# B&R Automation Studio project 305841_E00002_AM_0 (part 8)

#### ActionMotionFbs.st
```iecst
(********************************************************************
 * COPYRIGHT -- General Atomics
 ********************************************************************
 * Program: AxisStateMachine
 * File: ActionMoveVel.st
 * Author: Administrator
 * Created: January 22, 2014
 ********************************************************************
 * Implementation of program AxisStateMachine
 ********************************************************************)

ACTION ActionCallMotionFunctions:
  ActionMpAxisBasic;
  ActionCamInOut;
  ActionGearInOut;
  ActionOffsetShift;
  ActionPhaseShift;
END_ACTION

ACTION ActionMpAxisBasic:
  // 1) Range checks position, velocity, accel & Decel
  // 2) Packs the sMot_MoveParameters into a local axisBasicParamsStructure
  // 3) Detects parameter changes and manages the Update and UpdateDone bits
  // 4) Sets the fb command bits based on the axis sMot_AxisCommands structure
  // 5) Runs the fbMpAxisBasic funciton block
  // 6) Updates the axis structure with the status and axis info coming back from the fb

  // Make sure min/max values are not exceeded for position, velocity, accel, and decel.
  // Clamp if necessary

  // Position
  IF ax.MoveParameters.Position >  axPositionLimits.PositionLimitPos THEN
    ax.MoveParameters.Position :=  axPositionLimits.PositionLimitPos;
  END_IF;
  IF ax.MoveParameters.Position <  axPositionLimits.PositionLimitNeg THEN
    ax.MoveParameters.Position :=  axPositionLimits.PositionLimitNeg;
  END_IF;

  // Velocity
  IF ax.MoveParameters.Velocity > ax.MoveParameters.VelocityMax THEN
    ax.MoveParameters.Velocity := ax.MoveParameters.VelocityMax;
  END_IF;
  IF ax.MoveParameters.Velocity < ax.MoveParameters.VelocityMin THEN
    ax.MoveParameters.Velocity := ax.MoveParameters.VelocityMin;
  END_IF;

  // Accel and decel
  IF ax.MoveParameters.Acceleration > ax.MoveParameters.AccelMax THEN
    ax.MoveParameters.Acceleration := ax.MoveParameters.AccelMax;
  END_IF;
  IF ax.MoveParameters.Acceleration < ax.MoveParameters.AccelMin THEN
    ax.MoveParameters.Acceleration := ax.MoveParameters.AccelMin;
  END_IF;

  IF ax.MoveParameters.Deceleration > ax.MoveParameters.DecelMax THEN
    ax.MoveParameters.Deceleration := ax.MoveParameters.DecelMax;
  END_IF;
  IF ax.MoveParameters.Deceleration < ax.MoveParameters.DecelMin THEN
    ax.MoveParameters.Deceleration := ax.MoveParameters.DecelMin;
  END_IF;

  // The execution behavior is determined by the inputs set elsewhere
  // in particular the sMot_AxisCommands XxxxCmd bits,
  // and the values in sMot_MoveParameters structure

  // Axis reference set in init routine

  // Only enable the fb if the axis is not set to be ignored
  // TODO: Different check needed? Not sure how to tell if an axis reference is not set
  // It would be nice to check ax.fbMpAxisBasic.MpLink <> 0 for example, but this is a structure not an address
  IF NOT ax.Ignore AND ax.AxisNo <> 0 THEN
    ax.fbMpAxisBasic.Enable := TRUE;
  ELSE
    ax.fbMpAxisBasic.Enable := FALSE;
  END_IF;

  // Load the parameters from the sMot_MoveParameter structure into
  // local structure variables used for the fb
  fctPackMpAxisBasicParams(_I_UdtParams:= ADR(ax.MoveParameters), _IO_MpParams := axisBasicParams);

  // To allow move parameter changes to take effect without having to stop,
  // detect a difference between the desired parameters and the previous values.
  // If they are different, then set the update bit until the UpdateDone bit is set.
  // NOTE: This fb manages the ax.fbMpAxisCoupling.Update request and monitors the .UpdateDone bit
  // Use the .UpdateCouplingParams bit in the command structure if the application needs to control
  // when to trigger the update. If parameters need to be set in possibly different areas of the software,
  // and all the updates should take place at once, the update fb is called conditionally. The
  // checked bit can be set high so it is called all the time if the checked bit is not managed.
  ax.Commands.UpdateMoveParams:= TRUE;
  IF ax.Commands.UpdateMoveParams THEN
    ax.fbUpdateBFbParams(_IO_MpParams := axisBasicParams);
    ax.Commands.UpdateMoveParams := FALSE;
  END_IF;

  // TODO: Enforce move permissives

  // Use the commands from the axis structue
  ax.fbMpAxisBasic.ErrorReset := ax.Commands.DriveResetCmd;
  ax.fbMpAxisBasic.Power := ax.Commands.EnableCmd;
  ax.fbMpAxisBasic.Home := ax.Commands.HomeCmd;
  // There is no specific jog cmd. Use Move Velocity instead.
  ax.fbMpAxisBasic.MoveVelocity := ax.Commands.MoveVelocityCmd OR ax.Commands.MoveJogCmd;
  ax.fbMpAxisBasic.MoveAbsolute := ax.Commands.MoveAbsoluteCmd;
  ax.fbMpAxisBasic.MoveAdditive := ax.Commands.MoveRelativeCmd;
  ax.fbMpAxisBasic.Stop := ax.Commands.StopCmd;
  ax.fbMpAxisBasic.JogPositive := ax.Commands.MoveJogPositiveCmd;
  ax.fbMpAxisBasic.JogNegative := ax.Commands.MoveJogNegativeCmd;
  ax.fbMpAxisBasic.LimitLoad := ax.MoveParameters.EnableTorqueLimit;
  ax.fbMpAxisBasic.ReleaseBrake := ax.Commands.ReleaseBrakeCmd;
  ax.fbMpAxisBasic.AutoTune := FALSE; // TODO
  ax.fbMpAxisBasic.Simulate := FALSE; // TODO

  // Call the fb
  ax.fbMpAxisBasic();

  // Update the axis status structure
  ax.Status.Position := ax.fbMpAxisBasic.Position;
  ax.Status.Velocity := ax.fbMpAxisBasic.Velocity;
  ax.Status.IsPoweredOn := ax.fbMpAxisBasic.PowerOn;
  ax.Status.IsHomed := ax.fbMpAxisBasic.IsHomed;
  ax.Status.IsInVelocity := ax.fbMpAxisBasic.InVelocity;
  ax.Status.IsInPosition := ax.fbMpAxisBasic.InPosition;
  ax.Status.IsMoveActive := ax.fbMpAxisBasic.MoveActive;
  ax.Status.IsMoveDone := ax.fbMpAxisBasic.MoveDone;
  ax.Status.IsStopped := ax.fbMpAxisBasic.Stopped;
  ax.Status.IsTorqueLimitReady := ax.fbMpAxisBasic.LimitLoadReady;
  ax.Status.IsBrakeManuallyReleased := ax.fbMpAxisBasic.BrakeReleased;

  // Now load the sMot_AxisStatus structure with the data returned from the fb
  fctGetMpAxisInfo(_I_MpInfo := ADR(ax.fbMpAxisBasic.Info), _IO_UdtStatus := ax.Status);

  // Calculate special (algorithmic) positions
  CalcSpecialPositions;

  // Now that the status of this axis is known, copy it to the other axes slave status
  // area if this axis is specified as a slave.
  CopySlaveStatusToMaster;

END_ACTION

ACTION ActionCamInOut:
  // Execute the cam in or cam out fbs based on the CamIn/Out requests
  // The fbs are edge triggered, and the requests are cleared once serviced.
  // If the caming params change, another request must be made.
  // TODO: Is cam out and another cam in needed if params change?

  // Only execute the cam in fb if the axis number has been set,
  // the slave axis number has been set, and neither is set to be ignored,
  // and it is requested.
  IF ax.Ignore OR ax.AxisNo = AD_UNKNOWN OR
       ax.CouplingParameters.SlaveAxisNo = AD_UNKNOWN OR
       axes[ax.CouplingParameters.SlaveAxisNo].Ignore THEN
    // slave or master should be ignored
    // keep the requests and executes low
    ax.CouplingParameters.CamInReq := FALSE;
    ax.CouplingParameters.CamOutReq := FALSE;
    ax.fbCamIn.Execute := FALSE;
    ax.fbCamOut.Execute := FALSE;
  ELSIF ax.CouplingParameters.CamInReq THEN
    // CamIn request is made.
    // Clear the req so a future rising edge can be seen
    ax.CouplingParameters.CamInReq := FALSE;
    // Make sure the CamOut req and execute is clear
    ax.CouplingParameters.CamOutReq := FALSE;
    ax.fbCamOut.Execute := FALSE;
    // Load the cam in params, then set the execute input (edge triggered fb)
    ax.fbCamIn.MasterOffset := ax.CouplingParameters.CamMasterOffset;
    ax.fbCamIn.SlaveOffset := ax.CouplingParameters.CamSlaveOffset;
    ax.fbCamIn.MasterScaling := ax.CouplingParameters.CamScalingMaster;
    ax.fbCamIn.SlaveScaling := ax.CouplingParameters.CamScalingSlave;
    ax.fbCamIn.StartMode := ax.CouplingParameters.CamStartMode;
    ax.fbCamIn.MasterValueSource := ax.CouplingParameters.CamMasterValueSource;
    // force cam id 1 for now.
    ax.CouplingParameters.CamId := 1;
    ax.fbCamIn.CamID := ax.CouplingParameters.CamId;
    ax.fbCamIn.BufferMode := ax.CouplingParameters.CamBufferMode; // only mcAborting currently supported
    ax.fbCamIn.AdvancedParameters.Periodic := ax.CouplingParameters.CamIsPeriodic;
    ax.fbCamIn.AdvancedParameters.Velocity := 0.0; // disable, use (slave?) axis max vel
    ax.fbCamIn.AdvancedParameters.Acceleration := 0.0; // disable, use (slave?) axis max accel
    ax.fbCamIn.AdvancedParameters.Deceleration := 0.0; // disable, use (slave?) axis max decel
    ax.fbCamIn.AdvancedParameters.Jerk := 0.0; // only non-zero if using McProfGen
    ax.fbCamIn.Execute := TRUE; // fb looks for a rising edge
  ELSIF ax.CouplingParameters.CamOutReq THEN
    // Clear the req so a future rising edge can be seen
    ax.CouplingParameters.CamOutReq := FALSE;
    // Make sure the GearIn req and execute is clear
    ax.CouplingParameters.CamInReq := FALSE;
    ax.fbCamIn.Execute := FALSE;
    // Load the cam out params, then set the execute input (edge triggered fb)
    ax.fbCamOut.Jerk := 0.0; // only non-zero if using McProfGen
    ax.fbCamOut.Execute := TRUE;
  END_IF;

  // Call the cam in and cam out fbs.
  ax.fbCamIn();
  ax.fbCamOut();
  // Clear the exuecute bits. The fbs are edge triggerd, and would have been seen by the above call.
  ax.fbCamIn.Execute := FALSE;
  ax.fbCamOut.Execute := FALSE;

  // Update the axis status structure
  IF ax.fbCamIn.Active AND NOT ax.fbCamIn.Error THEN
    ax.Status.IsCamInSync := ax.fbCamIn.InSync;
    ax.Status.IsCamEndOfProfile := ax.fbCamIn.EndOfProfile;
    ax.Status.CamStatus := ax.fbCamIn.Status;
  ELSE
    ax.Status.IsCamInSync := FALSE;
    ax.Status.IsCamEndOfProfile := FALSE;
    ax.Status.CamStatus := mcCAM_STATUS_PREPARING_MOVE; // 0 value, but don't have a good choice for "not active
  END_IF;

END_ACTION

ACTION ActionGearInOut:
  // Execute the gear in or gear out fbs based on the GearIn/Out requests
  // The fbs are edge triggered, and the requests are cleared once serviced.
  // If the gearing params change, another request must be made.

  // Only execute the gear in fb if the axis number has been set,
  // the slave axis number has been set, and neither is set to be ignored,
  // and it is requested.
  IF ax.Ignore OR ax.AxisNo = AD_UNKNOWN OR
       ax.CouplingParameters.SlaveAxisNo = AD_UNKNOWN OR
       axes[ax.CouplingParameters.SlaveAxisNo].Ignore THEN
    // slave or master should be ignored
    // keep the requests and executes low
    ax.CouplingParameters.GearInReq := FALSE;
    ax.CouplingParameters.GearOutReq := FALSE;
    ax.fbGearIn.Execute := FALSE;
    ax.fbGearOut.Execute := FALSE;
  ELSIF ax.CouplingParameters.GearInReq THEN
    // GearIn request is made.
    // Clear the req so a future rising edge can be seen
    ax.CouplingParameters.GearInReq := FALSE;
    // Make sure the GearOut req and execute is clear
    ax.CouplingParameters.GearOutReq := FALSE;
    ax.fbGearOut.Execute := FALSE;
    // Load the gear in params, then set the execute input (edge triggered fb)
    ax.fbGearIn.RatioNumerator := ax.CouplingParameters.GearInRatioNumerator;
    ax.fbGearIn.RatioDenominator := ax.CouplingParameters.GearInRatioDenominator;
    ax.fbGearIn.MasterValueSource := ax.CouplingParameters.GearInMasterValueSource;
    ax.fbGearIn.Acceleration := ax.CouplingParameters.ShiftAccelerationMax;
    ax.fbGearIn.Deceleration := ax.CouplingParameters.ShiftDecelerationMax;
    ax.fbGearIn.Jerk := ax.CouplingParameters.ShiftJerk; // only non-zero if using McProfGen
    ax.fbGearIn.BufferMode := ax.CouplingParameters.GearInBufferMode; // onlly mcAborting currently supported
    ax.fbGearIn.AdvancedParameters.MasterMaxVelocity := ax.CouplingParameters.ShiftProfileBaseMaxVelocity;
    ax.fbGearIn.Execute := TRUE; // fb looks for a rising edge
  ELSIF ax.CouplingParameters.GearOutReq THEN
    // Clear the req so a future rising edge can be seen
    ax.CouplingParameters.GearOutReq := FALSE;
    // Make sure the GearIn req and execute is clear
    ax.CouplingParameters.GearInReq := FALSE;
    ax.fbGearIn.Execute := FALSE;
    // Load the gear out params, then set the execute input (edge triggered fb)
    ax.fbGearOut.Jerk := 0.0; // only non-zero if using McProfGen
    ax.fbGearOut.Execute := TRUE;
  END_IF;

  // Call the gear in and gear out fbs.
  ax.fbGearIn();
  ax.fbGearOut();
  // Clear the exuecute bits. The fbs are edge triggerd, and would have been seen by the above call.
  ax.fbGearIn.Execute := FALSE;
  ax.fbGearOut.Execute := FALSE;

  // Update the axis status structure.
  // Derrive InCompensation -- Active but not in sync
  IF ax.fbGearIn.Active AND NOT ax.fbGearIn.Error THEN
    // If gear in is active, it is either in sync or in compensation
    ax.Status.IsGearInSync := ax.fbGearIn.InGear;
    ax.Status.IsGearInCompensation := NOT ax.fbGearIn.InGear;
  ELSE
    ax.Status.IsGearInSync := FALSE;
    ax.Status.IsGearInCompensation := FALSE;
  END_IF;

END_ACTION

ACTION ActionOffsetShift:
  // Execute the offset shift fb based on the offset shift request.
  // The fb is edge triggered based on the StartShift input, however
  // either by design or because of a bug, the AdvancedParameters.ProfileBase
  // seems to be evaluated based on Enable going high, and chagese made after,
  // but before StartShift input going high are ignored.
  // If the offset params change, another request must be made.

  // Since triggering an offset while another offset is in progress triggers an error,
  // the request, enable, and start shift are only cleared once the shift is finished,
  // or the fb is invalid or in error

  // Only execute the offset shift fb if the axis number has been set,
  // the slave axis number has been set, and neither is set to be ignored,
  // and it is requested, and the master axis is powered (so enable can be easily toggled)
  IF ax.Ignore OR ax.AxisNo = AD_UNKNOWN OR
    ax.CouplingParameters.SlaveAxisNo = AD_UNKNOWN OR
    axes[ax.CouplingParameters.SlaveAxisNo].Ignore OR
    NOT ax.Status.IsPoweredOn THEN
    // slave or master should be ignored, or slave is not set, or
    // master is not powered.  Keep the request, enable, and startshift low
    ax.CouplingParameters.OffsetShiftReq := FALSE;
    ax.fbOffsetShift.Enable := FALSE;
    ax.fbOffsetShift.StartShift := FALSE;
  ELSIF ax.CouplingParameters.OffsetShiftReq AND NOT ax.fbOffsetShift.Enable THEN
    // Offset Shift request is made.
    // Set the fb params so a start shift can act on them. Set them
    // before bringing enable high because the profile base param(s) seem to
    // need to be set before the StartShift input is raised.
    ax.fbOffsetShift.OffsetShift := ax.CouplingParameters.Shift;
    ax.fbOffsetShift.Velocity := ax.CouplingParameters.ShiftVelocityMax;
    ax.fbOffsetShift.Acceleration := ax.CouplingParameters.ShiftAccelerationMax;
    ax.fbOffsetShift.AdvancedParameters.ShiftMode := ax.CouplingParameters.ShiftMode;
    ax.fbOffsetShift.AdvancedParameters.ProfileBase := ax.CouplingParameters.ShiftProfileBase;
    ax.fbOffsetShift.AdvancedParameters.ProfileBaseMaxVelocity := ax.CouplingParameters.ShiftProfileBaseMaxVelocity;
    ax.fbOffsetShift.AdvancedParameters.DistanceParameters.ProfileDistance := ax.CouplingParameters.ShiftProfileDistance;
    ax.fbOffsetShift.AdvancedParameters.ZoneParameters.StartPosition := ax.CouplingParameters.ShiftZoneStartPosition;
    ax.fbOffsetShift.AdvancedParameters.ZoneParameters.EndPosition := ax.CouplingParameters.ShiftZoneEndPosition;
    ax.fbOffsetShift.AdvancedParameters.ZoneParameters.Period := ax.CouplingParameters.ShiftZonePeriod;
    ax.fbOffsetShift.AdvancedParameters.ShiftAlternativeValueSource := mcALT_VALUE_NOT_USED;
    // Enable the fb so we can look for a valid before starting the shift.
    ax.fbOffsetShift.Enable := TRUE;
  ELSIF ax.CouplingParameters.OffsetShiftReq AND ax.fbOffsetShift.Enable AND
    NOT ax.fbOffsetShift.StartShift AND ax.fbOffsetShift.Valid AND NOT ax.fbOffsetShift.Error THEN
    // fb is enabled and valid and not in error, but not started yet.
    // Start the shift on the edge triggered StartShift input.
    ax.fbOffsetShift.StartShift := TRUE;
  ELSIF ax.CouplingParameters.OffsetShiftReq AND ax.fbOffsetShift.Enable AND
    (NOT ax.fbOffsetShift.Valid AND ax.fbOffsetShift.Error) THEN
    // fb is enabled but not valid or in error. Clear the request, enable, and make sure the start shift stays low
    ax.CouplingParameters.OffsetShiftReq := FALSE;
    ax.fbOffsetShift.Enable := FALSE;
    ax.fbOffsetShift.StartShift := FALSE;
  ELSIF ax.CouplingParameters.OffsetShiftReq AND ax.fbOffsetShift.Valid AND ax.fbOffsetShift.StartShift AND
    NOT ax.fbOffsetShift.ShiftAttained THEN
    // Shift was triggered, but isn't done yet.
    // Update the axis status structure
    ax.Status.IsCoordOffsetShiftAttained := FALSE;
    ax.Status.IsCoordOffsetShiftStarted := ax.fbOffsetShift.ShiftStarted;
    ax.Status.CoordActualOffsetShift := ax.fbOffsetShift.ActualOffsetShift;
  ELSIF ax.CouplingParameters.OffsetShiftReq AND ax.fbOffsetShift.Valid AND ax.fbOffsetShift.StartShift AND
    ax.fbOffsetShift.ShiftAttained THEN
    // Shift was triggered, and is now done.
    // Update the axis status structure
    ax.Status.IsCoordOffsetShiftAttained := ax.fbOffsetShift.ShiftAttained;
    ax.Status.IsCoordOffsetShiftStarted := FALSE;
    ax.Status.CoordActualOffsetShift := ax.fbOffsetShift.ActualOffsetShift;
    // Clear the request, enable, and start shift.
    // Clearing the original request at the end prevents another request from triggering a shift while
    // a shift is in progress, but also allows another request to be triggered once done.
    ax.CouplingParameters.OffsetShiftReq := FALSE;
    ax.fbOffsetShift.Enable := FALSE;
    ax.fbOffsetShift.StartShift := FALSE;
  END_IF;

  // Call the offset shift fb.
  ax.fbOffsetShift();

END_ACTION

ACTION ActionPhaseShift:
  // Execute the phase shift fb based on the phase shift request.
  // The fb is edge triggered, and the request is cleared once serviced.
  // If the phase params change, another request must be made.
  // TODO: Verify operation/behavior when changing params

  // Only execute the phase shift fb if the axis number has been set,
  // the slave axis number has been set, and neither is set to be ignored,
  // and it is requested, and the master axis is powered (so enable can be easily toggled)
  IF ax.Ignore OR ax.AxisNo = AD_UNKNOWN OR
       ax.CouplingParameters.SlaveAxisNo = AD_UNKNOWN OR
       axes[ax.CouplingParameters.SlaveAxisNo].Ignore OR
       NOT ax.Status.IsPoweredOn THEN
    // slave or master should be ignored
    // keep the request and enable low
    ax.CouplingParameters.PhaseShiftReq := FALSE;
    ax.fbPhaseShift.Enable := FALSE;
    ax.fbPhaseShift.StartShift := FALSE;
  ELSE
    ax.fbPhaseShift.Enable := TRUE;
  END_IF;

  // Enable input and ignore considered above. If req is high,
  // it can be acted upon.
  IF ax.CouplingParameters.PhaseShiftReq THEN
    // Phase Shift request is made.
    // Clear the req so a future rising edge can be seen
    ax.CouplingParameters.PhaseShiftReq := FALSE;
    // Load the phase shift params, then set the start shift input (edge sensitive input)
    ax.fbPhaseShift.PhaseShift := ax.CouplingParameters.Shift;
    ax.fbPhaseShift.Velocity := ax.CouplingParameters.ShiftVelocityMax;
    ax.fbPhaseShift.Acceleration := ax.CouplingParameters.ShiftAccelerationMax;
    ax.fbPhaseShift.AdvancedParameters.ShiftMode := ax.CouplingParameters.ShiftMode;
    ax.fbPhaseShift.AdvancedParameters.ProfileBase := ax.CouplingParameters.ShiftProfileBase;
    ax.fbPhaseShift.AdvancedParameters.ProfileBaseMaxVelocity := ax.CouplingParameters.ShiftProfileBaseMaxVelocity;
    ax.fbPhaseShift.AdvancedParameters.DistanceParameters.ProfileDistance := ax.CouplingParameters.ShiftProfileDistance;
    ax.fbPhaseShift.AdvancedParameters.ZoneParameters.StartPosition := ax.CouplingParameters.ShiftZoneStartPosition;
    ax.fbPhaseShift.AdvancedParameters.ZoneParameters.EndPosition := ax.CouplingParameters.ShiftZoneEndPosition;
    ax.fbPhaseShift.AdvancedParameters.ZoneParameters.Period := ax.CouplingParameters.ShiftZonePeriod;
    ax.fbPhaseShift.AdvancedParameters.ShiftAlternativeValueSource := mcALT_VALUE_NOT_USED;
    ax.fbPhaseShift.StartShift := TRUE; // fb looks for a rising edge
  END_IF;

  // Call the phase shift fb.
  ax.fbPhaseShift();
  // Clear the start shift bit. The fb is edge triggerd, and it would have been seen by the above call.
  ax.fbPhaseShift.StartShift := FALSE; // fb looks for a rising edge

  // Update the axis status structure as long as status is valid and there is no error.
  // Otherwise, clear the values
  IF ax.fbPhaseShift.Valid AND NOT ax.fbPhaseShift.Error THEN
    ax.Status.IsCoordPhaseShiftAttained := ax.fbPhaseShift.ShiftAttained;
    ax.Status.IsCoordPhaseShiftStarted := ax.fbPhaseShift.ShiftStarted;
    ax.Status.CoordActualPhaseShift := ax.fbPhaseShift.ActualPhaseShift;
  ELSE
    ax.Status.IsCoordPhaseShiftAttained := FALSE;
    ax.Status.IsCoordPhaseShiftStarted := FALSE;
    ax.Status.CoordActualPhaseShift := 0.0;
  END_IF;

END_ACTION

ACTION CopySlaveStatusToMaster :
  // If this axis number is a slave to another axis, then copy this axis
  // status to the master axis structure. This is a convenience
  // so the HMI for example, only needs to look in one structure (the master) and
  // can access the slave status.

  // Loop thru the axes. If the axis of index has this axis specified as a slave axis,
  // copy this axis status to the axis of index slave status.
  // Axis 0 is a dummy axis, so it can be skipped.
  FOR axIdx := 1 TO AXIS_COUNT DO
    IF axes[axIdx].CouplingParameters.SlaveAxisNo = AXIS_NO THEN
      // This axis is a slave to the axis referenced by axIdx.
      // Copy this axis status to the indexed axis slave status
      fctCopyAxisStatus(_I_SrcStatus := ADR(ax.Status), _I_DestStatus := ADR(axes[axIdx].StatusSlave));
    END_IF;
  END_FOR;
END_ACTION
```

#### AxSMCyclic - Copy.sfc
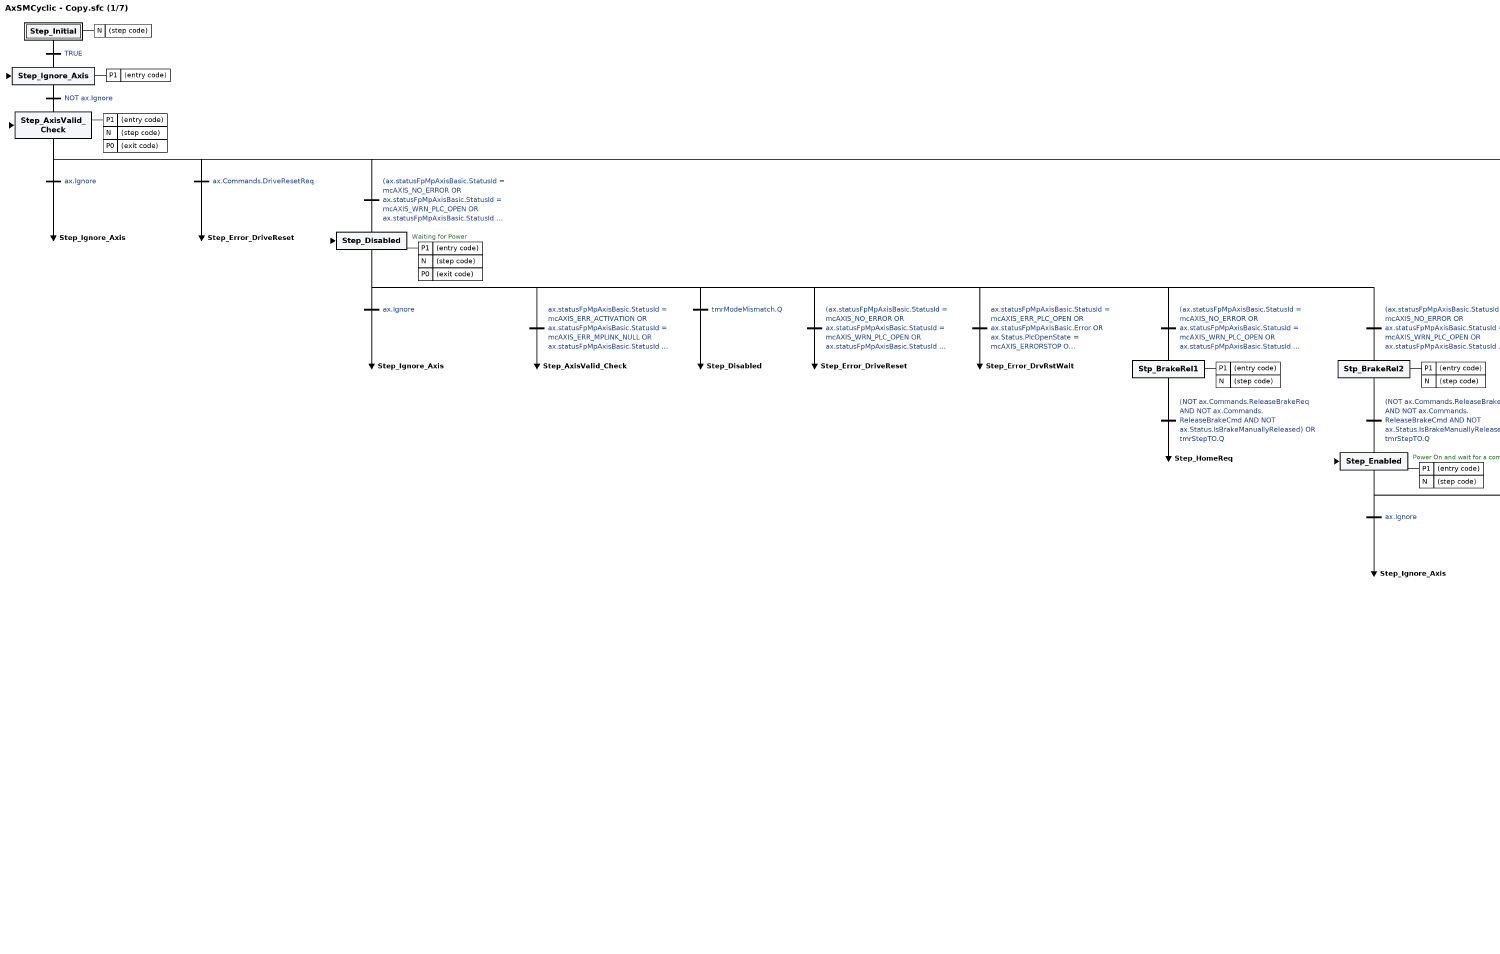
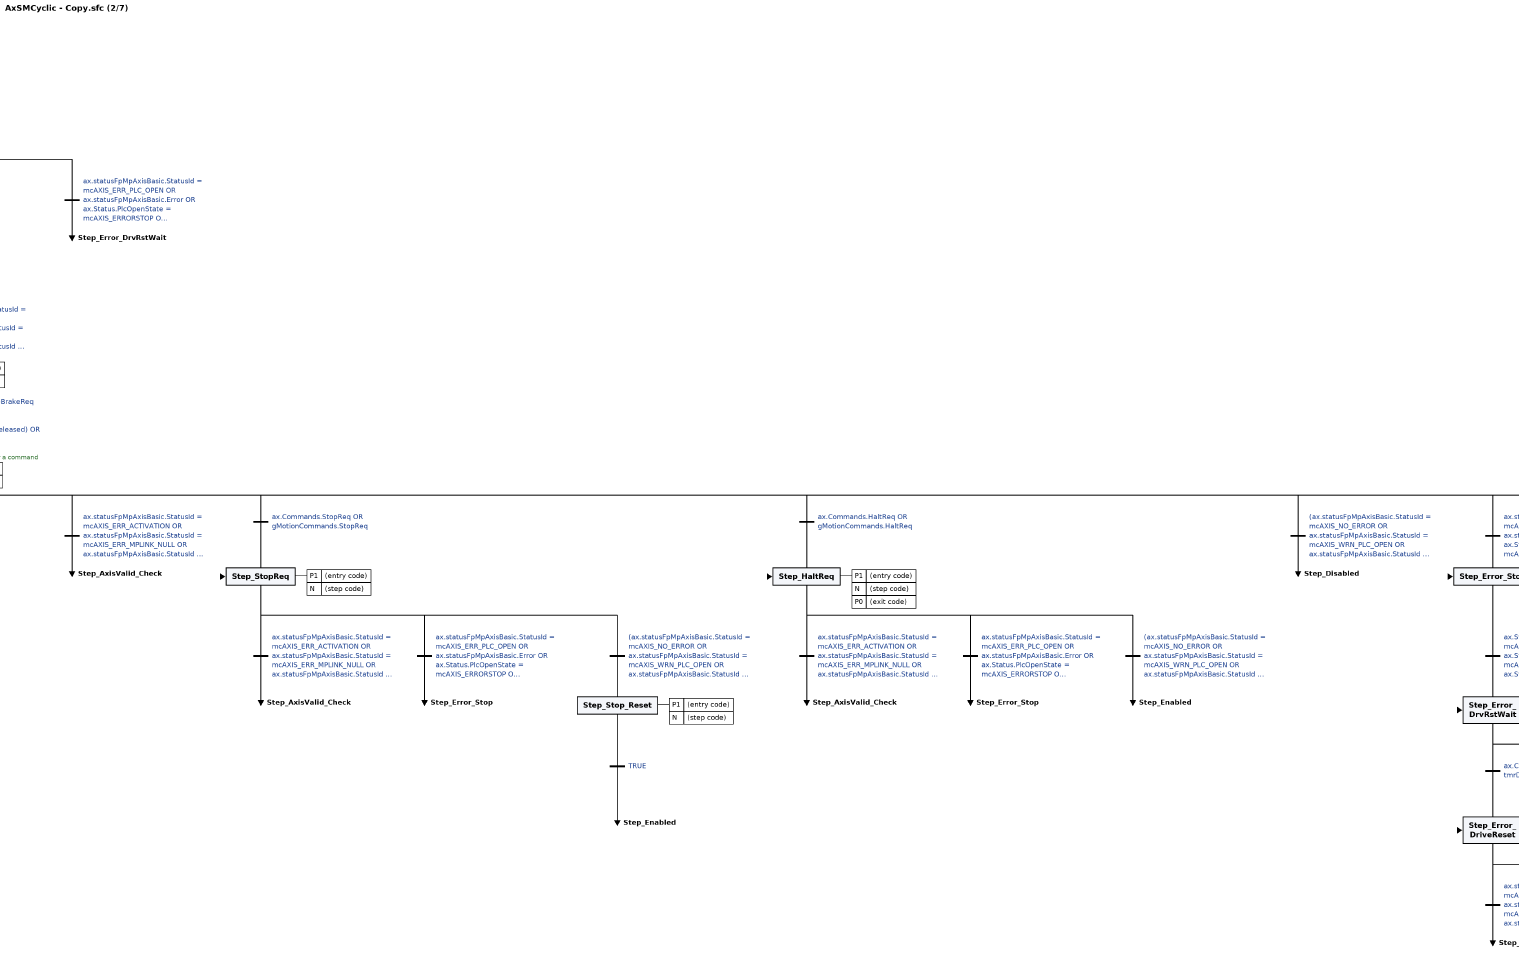
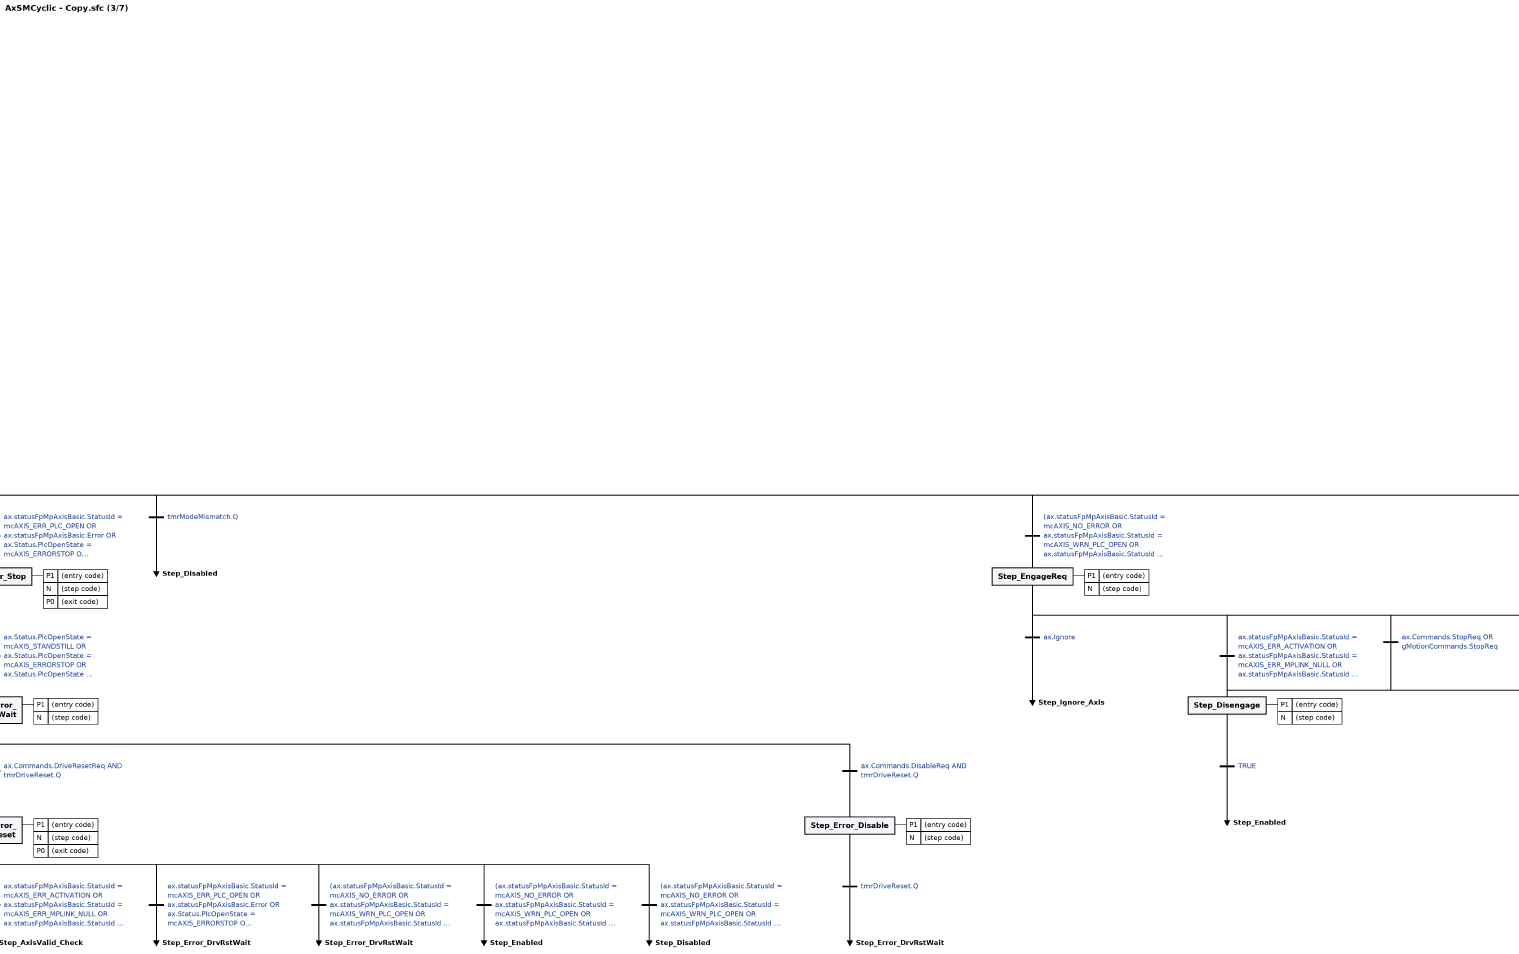
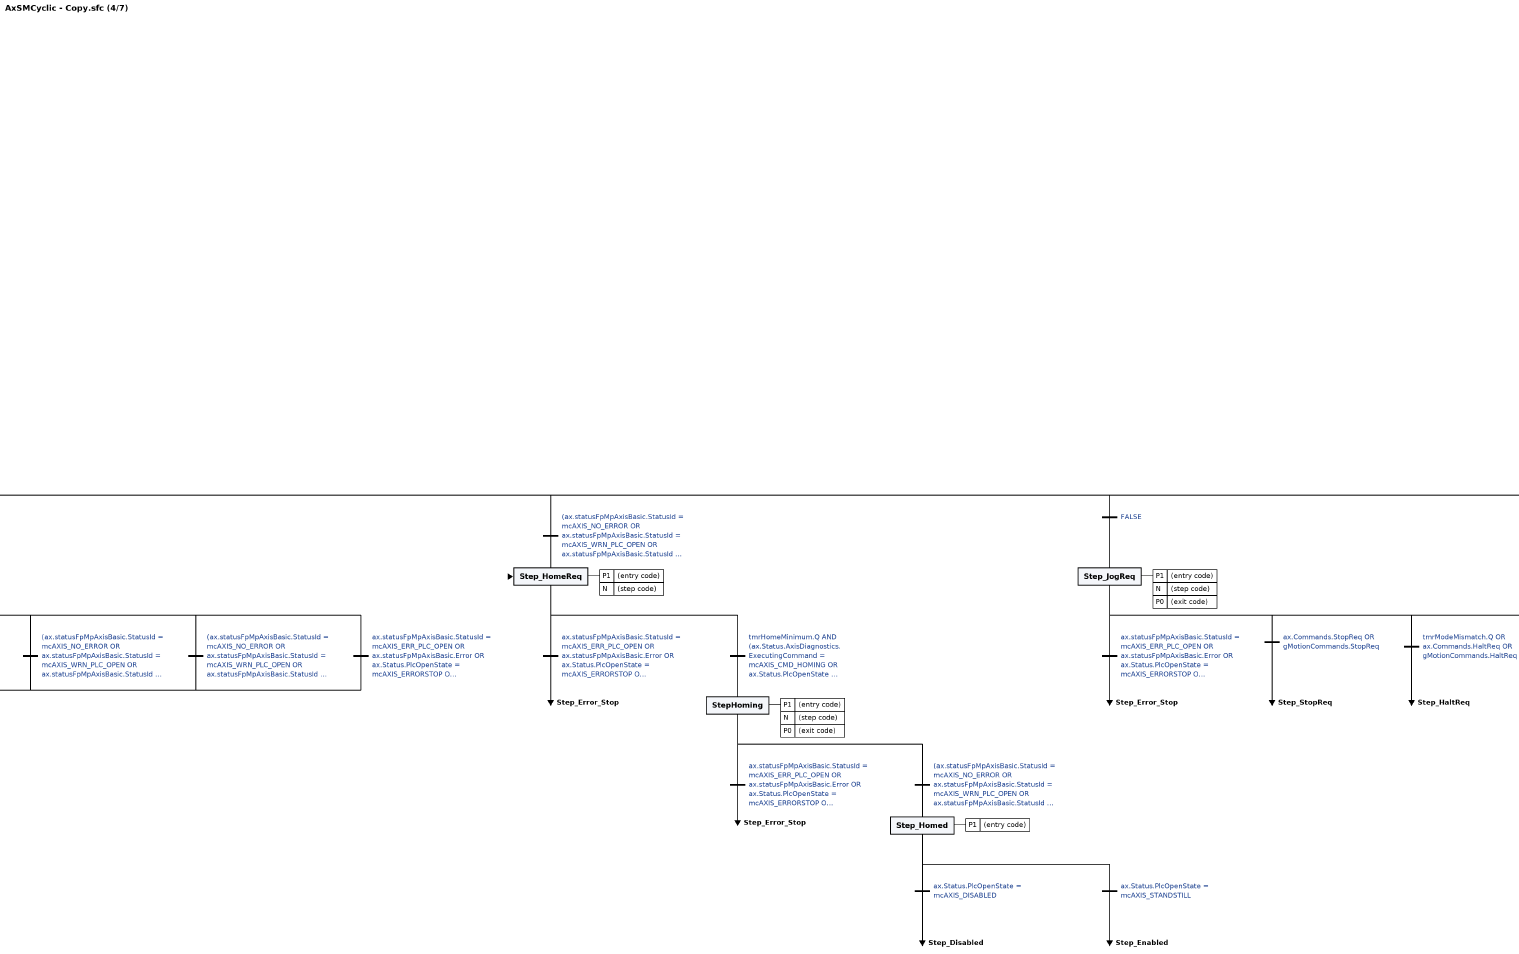
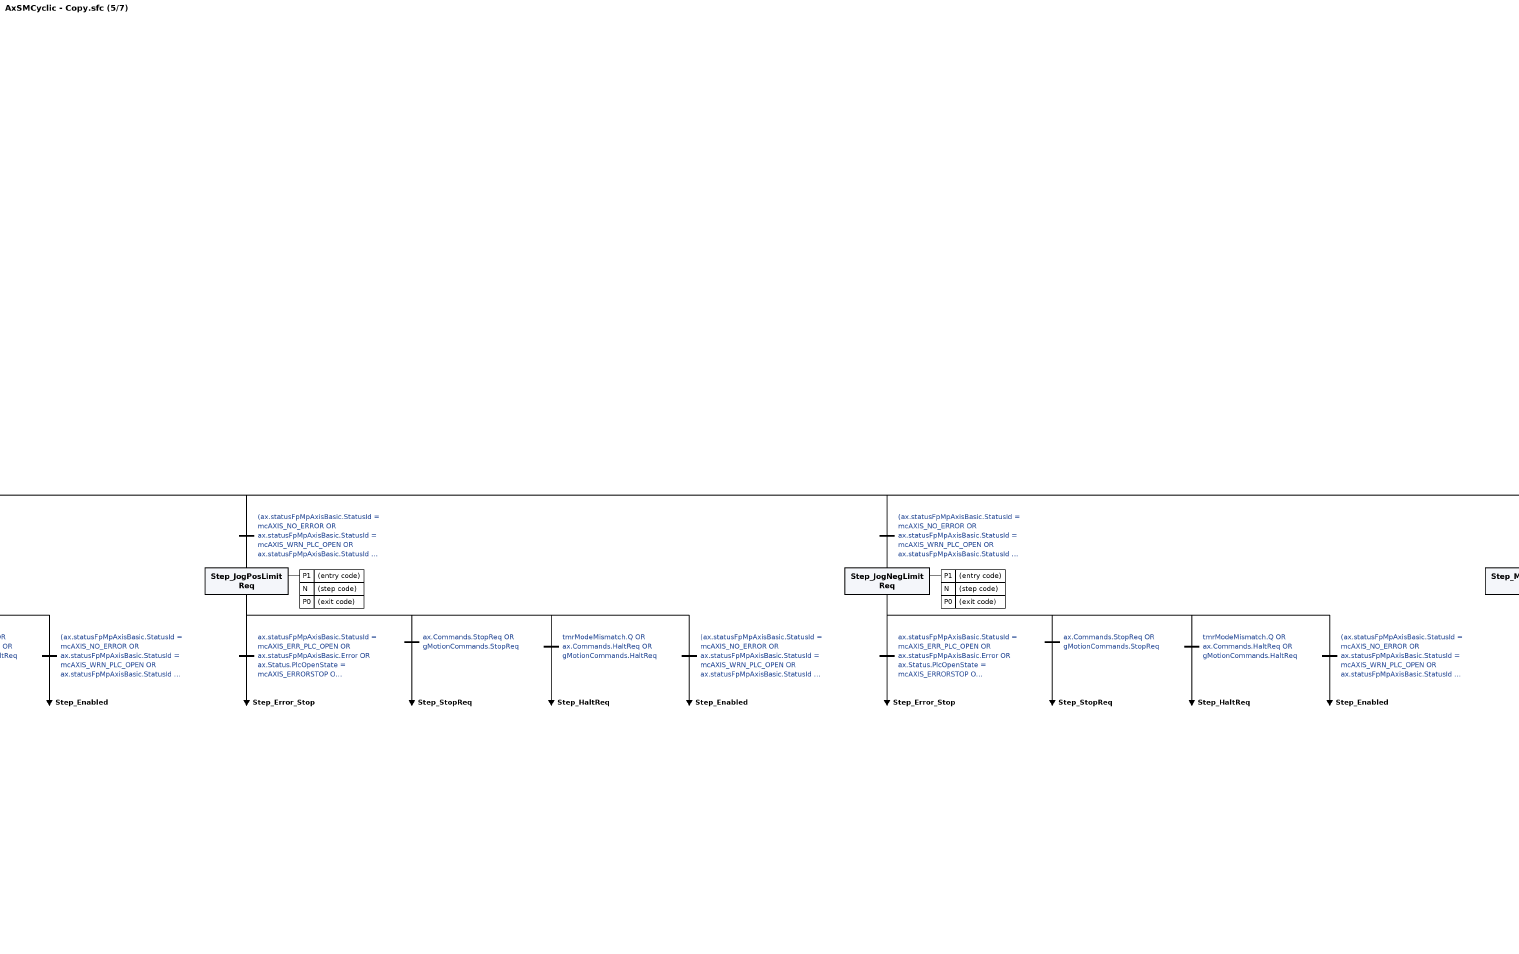
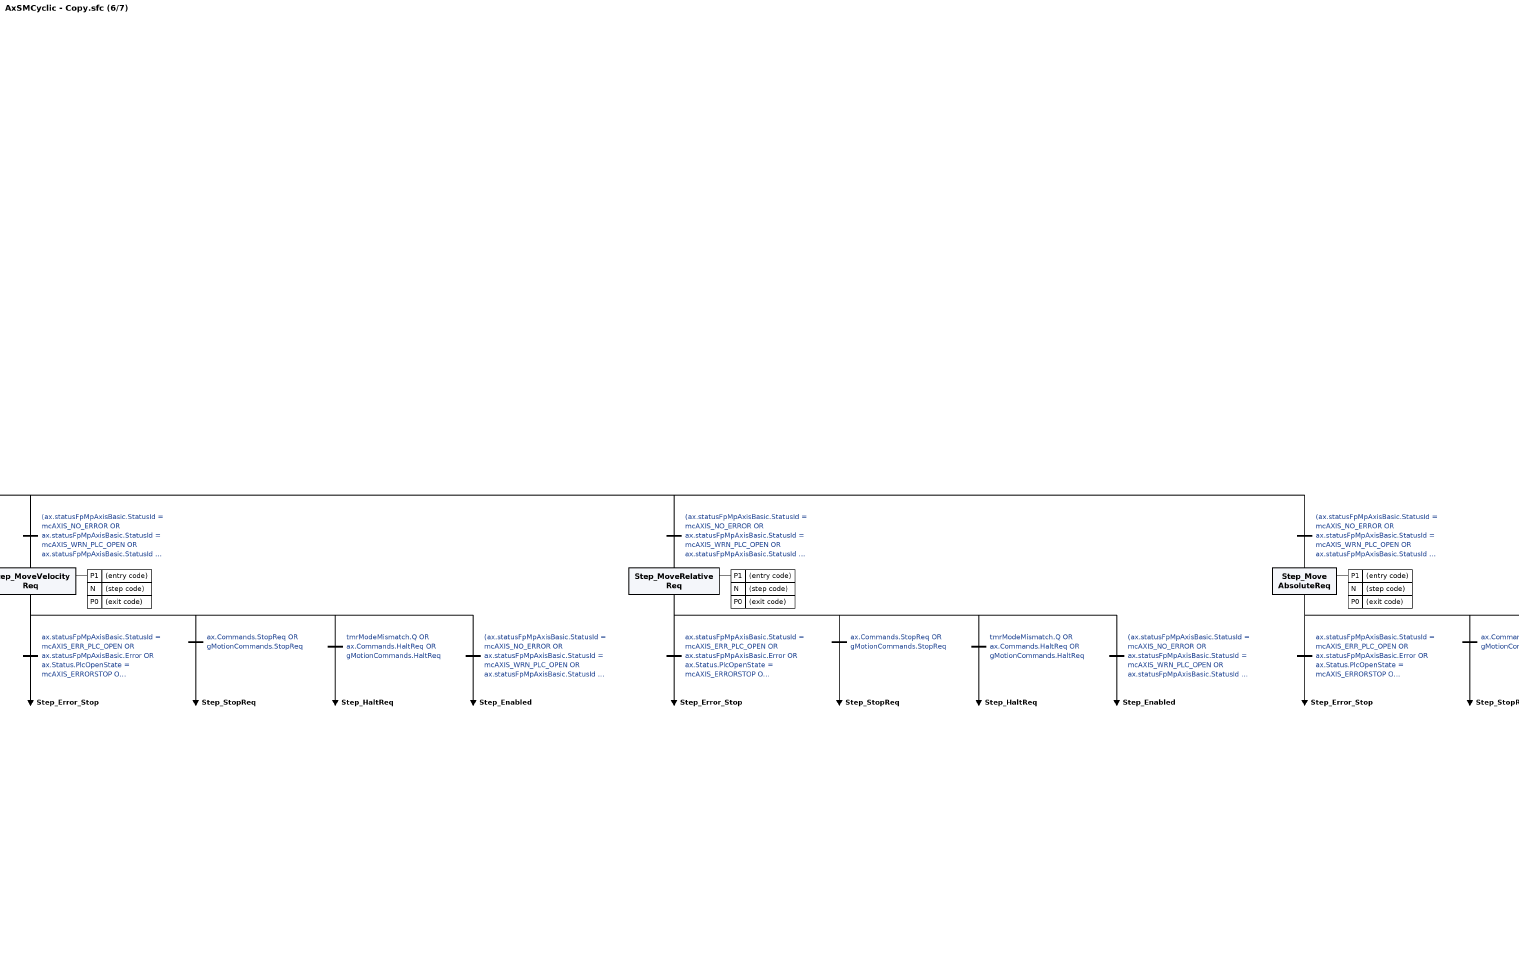
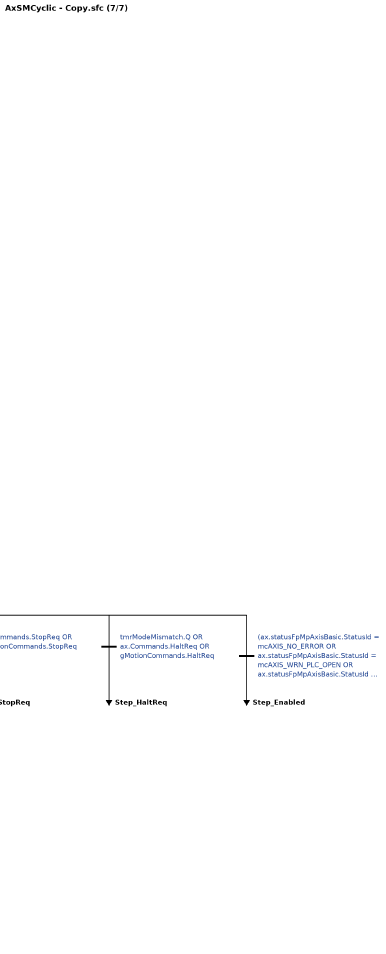
```iecst
PROGRAM _CYCLIC
INITIAL_STEP Step_Initial:
// Set the state
ax.SMState:= GAMOT_ASMS_INITIAL;

// Most stuff initialized in the AxSMInit.st routine

// init drive reset delay timer
tmrDriveReset.PT:= T#5s;

END_STEP
TRANSITION FROM Step_Initial TO Step_Ignore_Axis:=
TRUE
END_TRANSITION
STEP Step_Ignore_Axis:
END_STEP
ENTRY_ACTION
// Set the state
ax.SMState:= GAMOT_ASMS_IGNORE;

END_ACTION
TRANSITION FROM Step_Ignore_Axis TO Step_AxisValid_Check:=
NOT ax.Ignore
END_TRANSITION
STEP Step_AxisValid_Check:
// Clear the commands and run MpAxisBasic to get status
// From this state, you can only get to the ignore, disable, or error states,
// but the transition to ignore, disable, or error happens without operator requests,
// so no need to consider any requests.

fctClearMotionCommands(_I_CmdMask := MACM_NOMASK, _IO_Commands := ax.Commands);
fctClearMotionRequests(_I_ReqMask := MACM_NOMASK, _IO_Commands := ax.Commands);
ActionCallMotionFunctions;

// If the axis in invalid, periodically run the fb with the input disabled to
// force a rising edge the next time.
tmrDriveReset(IN:= ax.statusFpMpAxisBasic.StatusId <> mcAXIS_NO_ERROR AND NOT tmrDriveReset.Q);
IF (tmrDriveReset.Q) THEN
  ax.fbMpAxisBasic(Enable:= FALSE);
END_IF;
END_STEP
ENTRY_ACTION
// Set the state
ax.SMState:= GAMOT_ASMS_VALID_CHECK;
END_ACTION
EXIT_ACTION
// Reset the drive reset timer
tmrDriveReset(IN:= FALSE);
END_ACTION
TRANSITION FROM Step_AxisValid_Check TO Step_Ignore_Axis:=
ax.Ignore
END_TRANSITION
(* @SFCISJUMP := 'Step_Ignore_Axis' *)
TRANSITION Reset Req FROM Step_AxisValid_Check TO Step_Error_DriveReset:=
// Drive reset request
ax.Commands.DriveResetReq

END_TRANSITION
(* @SFCISJUMP := 'Step_Error_DriveReset' *)
TRANSITION Valid and no errors FROM Step_AxisValid_Check TO Step_Disabled:=
// Valid status (allow the couple axis warnings), and no errors
(ax.statusFpMpAxisBasic.StatusId = mcAXIS_NO_ERROR OR
ax.statusFpMpAxisBasic.StatusId = mcAXIS_WRN_PLC_OPEN OR
ax.statusFpMpAxisBasic.StatusId = mcAXIS_WRN_MULTIPLE_COMMAND) AND
NOT ax.statusFpMpAxisBasic.Error
END_TRANSITION
STEP Step_Disabled:
// From the disabled state, you can only get to
// the Ready (enabled/powered), Home, Error, or drive reset states,
// but this state does not send any commands, except for the brake release if requested.
// Clear all the commands except for brake release.
// Allow the Enable, Brake Release, Home, and Reset requests
// Note: The brake release is only valid in this state. This command will get cleared when leaving this state
fctClearMotionCommands(_I_CmdMask := MACM_RELEASE_BRAKE_MASK, _IO_Commands := ax.Commands);

// Set the release brake command if requested. Give priority to the clear cmd.
IF  ax.Commands.ClearReleaseBrakeReq THEN
  ax.Commands.ReleaseBrakeCmd := FALSE;
ELSIF ax.Commands.ReleaseBrakeReq THEN
  ax.Commands.ReleaseBrakeCmd := TRUE;
END_IF;

// Call motion command to get status and possibly release the brake
ActionCallMotionFunctions;

// Clear the requests other than the enable, home, and drive reset
reqMask := MACM_ENABLE_MASK + MACM_HOME_MASK + MACM_DRIVE_RESET_MASK;
fctClearMotionRequests(_I_ReqMask := reqMask, _IO_Commands := ax.Commands);

// Run the mode mismatch timer if the mode is not ok.
// Assume mode is okay - no modes on this system
tmrModeMismatch(IN:= FALSE);
END_STEP
(* @SFCCOMMENT := 'Waiting for Power' *)
ENTRY_ACTION
// Set the state
ax.SMState:= GAMOT_ASMS_DISABLED;
END_ACTION
EXIT_ACTION
// On exit, clear the the brake release cmd and requests since they are only valid in this state.
ax.Commands.ReleaseBrakeReq := FALSE;
ax.Commands.ClearReleaseBrakeReq := FALSE;
ax.Commands.ReleaseBrakeCmd := FALSE;
END_ACTION
TRANSITION FROM Step_Disabled TO Step_Ignore_Axis:=
ax.Ignore
END_TRANSITION
(* @SFCISJUMP := 'Step_Ignore_Axis' *)
TRANSITION Invalid Status FROM Step_Disabled TO Step_AxisValid_Check:=
ax.statusFpMpAxisBasic.StatusId = mcAXIS_ERR_ACTIVATION OR
ax.statusFpMpAxisBasic.StatusId = mcAXIS_ERR_MPLINK_NULL OR
ax.statusFpMpAxisBasic.StatusId = mcAXIS_ERR_MPLINK_INVALID OR
ax.statusFpMpAxisBasic.StatusId = mcAXIS_ERR_MPLINK_CHANGED OR
ax.statusFpMpAxisBasic.StatusId = mcAXIS_ERR_MPLINK_CORRUPT OR
ax.statusFpMpAxisBasic.StatusId = mcAXIS_ERR_MPLINK_IN_USE OR
ax.statusFpMpAxisBasic.StatusId = mcAXIS_ERR_PAR_NULL
END_TRANSITION
(* @SFCISJUMP := 'Step_AxisValid_Check' *)
TRANSITION Mode problem FROM Step_Disabled TO Step_Disabled:=
// mode mismatch timer times out
tmrModeMismatch.Q
END_TRANSITION
(* @SFCISJUMP := 'Step_Disabled' *)
TRANSITION no errors, reset req FROM Step_Disabled TO Step_Error_DriveReset:=
// Valid status (allow the couple axis warnings), no errors, drive reset req
(ax.statusFpMpAxisBasic.StatusId = mcAXIS_NO_ERROR OR
ax.statusFpMpAxisBasic.StatusId = mcAXIS_WRN_PLC_OPEN OR
ax.statusFpMpAxisBasic.StatusId = mcAXIS_WRN_MULTIPLE_COMMAND) AND
NOT ax.statusFpMpAxisBasic.Error AND
ax.Commands.DriveResetReq
END_TRANSITION
(* @SFCISJUMP := 'Step_Error_DriveReset' *)
TRANSITION valid but error FROM Step_Disabled TO Step_Error_DrvRstWait:=
// Valid status, but an error
ax.statusFpMpAxisBasic.StatusId = mcAXIS_ERR_PLC_OPEN OR
ax.statusFpMpAxisBasic.Error OR
ax.Status.PlcOpenState = mcAXIS_ERRORSTOP OR
ax.Status.PlcOpenState = mcAXIS_INVALID_CONFIGURATION
END_TRANSITION
(* @SFCISJUMP := 'Step_Error_DrvRstWait' *)
TRANSITION no errors, home req FROM Step_Disabled TO Stp_BrakeRel1:=
// Valid status (allow the couple axis warnings), no errors, home request
(ax.statusFpMpAxisBasic.StatusId = mcAXIS_NO_ERROR OR
ax.statusFpMpAxisBasic.StatusId = mcAXIS_WRN_PLC_OPEN OR
ax.statusFpMpAxisBasic.StatusId = mcAXIS_WRN_MULTIPLE_COMMAND) AND
NOT ax.statusFpMpAxisBasic.Error AND
ax.Commands.HomeReq
END_TRANSITION
STEP Stp_BrakeRel1:
// On the way to homeing, but not there yet ... Need to make sure the manual brake release is off
// Clear all the commands.
// Allow the Home request since that is where we are going
fctClearMotionCommands(_I_CmdMask := MACM_NOMASK, _IO_Commands := ax.Commands);
fctClearMotionRequests(_I_ReqMask := MACM_HOME_MASK, _IO_Commands := ax.Commands);

// Call motion command to get status and possibly release the brake
ActionCallMotionFunctions;

// Run step TO timer
tmrStepTO(IN:= TRUE);
END_STEP
ENTRY_ACTION
// Reset step TO tmr
tmrStepTO(IN:= FALSE, PT:= T#500ms);
END_ACTION
TRANSITION brake off or TO FROM Stp_BrakeRel1 TO Step_HomeReq:=
// Manual brake release should turn off, but don't allow us to get stuck here.
// Errors will be caught once in the home state.
(NOT ax.Commands.ReleaseBrakeReq AND
NOT ax.Commands.ReleaseBrakeCmd AND
NOT ax.Status.IsBrakeManuallyReleased)
OR
tmrStepTO.Q
END_TRANSITION
(* @SFCISJUMP := 'Step_HomeReq' *)
TRANSITION no errors, global or axis enable req FROM Step_Disabled TO Stp_BrakeRel2:=
// // Valid status (allow the couple axis warnings), no errors and enable req or global enable req
// TODO: How to deal with handling global request (local OS or some sort or reset of cmd)
(ax.statusFpMpAxisBasic.StatusId = mcAXIS_NO_ERROR OR
ax.statusFpMpAxisBasic.StatusId = mcAXIS_WRN_PLC_OPEN OR
ax.statusFpMpAxisBasic.StatusId = mcAXIS_WRN_MULTIPLE_COMMAND) AND
NOT ax.statusFpMpAxisBasic.Error AND
(ax.Commands.EnableReq OR gMotionCommands.EnableReq)
END_TRANSITION
STEP Stp_BrakeRel2:
// On the way to enable, but not there yet ... Need to make sure the manual brake release is off
// Clear all the commands.
// Allow the Enable request since that is where we are going
fctClearMotionCommands(_I_CmdMask := MACM_NOMASK, _IO_Commands := ax.Commands);
fctClearMotionRequests(_I_ReqMask := MACM_ENABLE_MASK, _IO_Commands := ax.Commands);

// Call motion command to get status and possibly release the brake
ActionCallMotionFunctions;

// Run step TO timer
tmrStepTO(IN:= TRUE);
END_STEP
ENTRY_ACTION
// Reset step TO tmr
tmrStepTO(IN:= FALSE, PT:= T#500ms);
END_ACTION
TRANSITION brake off or TO FROM Stp_BrakeRel2 TO Step_Enabled:=
// Manual brake release should turn off, but don't allow us to get stuck here.
// Errors will be caught once in the enable state.
(NOT ax.Commands.ReleaseBrakeReq AND
NOT ax.Commands.ReleaseBrakeCmd AND
NOT ax.Status.IsBrakeManuallyReleased)
OR
tmrStepTO.Q
END_TRANSITION
STEP Step_Enabled:
// From the enabled state, you get to
// the error, home, stop, halt, engage, move or disabled states.
// This state will honor the above listed requests.
// This state will send a power command.
// You might get here from another move command if a move request comes in for a move during another move,
// so to prevent a bump when honoring a new move request, don't indiscriminently clear the commands.
ax.Commands.EnableCmd := TRUE;

// Jog no used with MpAxisBasic. Velocity move or jog positive limit or jog negative limit used in place of jog.
// Replace a jog request with a velocity req.
ax.Commands.MoveVelocityReq := ax.Commands.MoveVelocityReq OR ax.Commands.MoveJogReq;
ax.Commands.MoveJogReq := FALSE;
ax.Commands.MoveJogCmd := FALSE;

// Initialize the req mask. This will be used at the bottom to clear the other (unwanted) requests.
// In between, however, allowed requests may modify the mask.
reqMask := MACM_DISABLE_MASK + MACM_HOME_MASK + MACM_STOP_MASK + MACM_HALT_MASK;

// Qualify move requests
  // Upon a request, check permissives.
  // If the not allowed flag is clear, then allow the move
  // and clear the other requests.
  // The order of the request checks give priority as follows
  // jog, jog limit positive, jog limit negative, velocity, relative, absolute, engage slave, disengage slave
  // The above priority is somewhat arbitrary, but an order was needed, because only one
  // move is allowed, and each move clears the other requests.  There may be a better/more sensical priority, however.

// Jog Command
IF ax.Commands.MoveJogReq THEN
  ActionChkPermissiveContinuous;
  IF (ax.Commands.MoveNotAllowed OR NOT ax.Status.IsHomed OR ax.ForceSetRef) THEN
    // Move not allowed in requested direction or axis is not homed, or it needs to be re-referenced
    // Set the mask to clear the request, preserving disable, halt and stop reqs
    // Mask set above, nothing to do
    // reqMask := MACM_DISABLE_MASK + MACM_STOP_MASK + MACM_HALT_MASK;
    ;
  ELSE
    // Move allowed, leave the request
    // Modify the mask set above, and clear the other move requests, preserving disable, halt and stop reqs
    reqMask := reqMask + MACM_JOG_MASK;
  END_IF
END_IF

// Jog Positive Limit Request
// Jog Limit requires move permissives.  The FB
// checks the position window, so this is a duplication of the
// application position window check.
IF ax.Commands.MoveJogPositiveReq THEN
  ActionChkPermissiveContinuous;
  IF (ax.Commands.MoveNotAllowed OR NOT ax.Status.IsHomed OR ax.ForceSetRef) THEN
    // Move not allowed in requested direction or axis is not homed, or it needs to be re-referenced
    // Set the mask to clear the request, preserving disable, halt and stop reqs
    // Mask set above, nothing to do
    // reqMask := MACM_DISABLE_MASK + MACM_STOP_MASK + MACM_HALT_MASK;
    ;
  ELSE
    // Move allowed, leave the request
    // Modify the mask set above, and clear the other move requests, preserving disable, halt and stop reqs
    reqMask := reqMask + MACM_JOG_POSITIVE_MASK;
  END_IF
END_IF

// Jog Negative Limit Request
// Jog Limit requires move permissives.  The FB
// checks the position window, so this is a duplication of the
// application position window check.
IF ax.Commands.MoveJogNegativeReq THEN
  ActionChkPermissiveContinuous;
  IF (ax.Commands.MoveNotAllowed OR NOT ax.Status.IsHomed OR ax.ForceSetRef) THEN
    // Move not allowed in requested direction or axis is not homed, or it needs to be re-referenced
    // Set the mask to clear the request, preserving disable, halt and stop reqs
    // Mask set above, nothing to do
    // reqMask := MACM_DISABLE_MASK + MACM_STOP_MASK + MACM_HALT_MASK;
    ;
  ELSE
    // Move allowed, leave the request
    // Modify the mask set above, and clear the other move requests, preserving disable, halt and stop reqs
    reqMask := reqMask + MACM_JOG_NEGATIVE_MASK;
  END_IF
END_IF

// Move Velocity Request
IF ax.Commands.MoveVelocityReq THEN
  // Take a snapshot of the current position.
  // This is to allow permissive checking while on the move
  // and while supporting a changealbe move window
  ax.MoveParameters.PermissiveCheck.StartPosition:= ax.Status.Position;
  ActionChkPermissiveRel;
  IF (ax.Commands.MoveNotAllowed OR NOT ax.Status.IsHomed OR ax.ForceSetRef) THEN
    // Move not allowed in requested direction or axis is not homed, or it needs to be re-referenced
    // Set the mask to clear the request, preserving disable, halt and stop reqs
    // Mask set above, nothing to do
    // reqMask := MACM_DISABLE_MASK + MACM_STOP_MASK + MACM_HALT_MASK;
    ;
  ELSE
    // Move allowed, leave the request
    // Modify the mask set above, and clear the other move requests, preserving disable, halt and stop reqs
    reqMask := reqMask + MACM_VELOCITY_MOVE_MASK;
  END_IF
END_IF

// Move Relative Request
IF ax.Commands.MoveRelativeReq THEN
  // Take a snapshot of the current position.
  // This is to allow permissive checking while on the move
  // and while supporting a changealbe move window
  ax.MoveParameters.PermissiveCheck.StartPosition:= ax.Status.Position;
  ActionChkPermissiveRel;
  IF (ax.Commands.MoveNotAllowed OR NOT ax.Status.IsHomed OR ax.ForceSetRef) THEN
    // Move not allowed in requested direction or axis is not homed, or it needs to be re-referenced
    // Set the mask to clear the request, preserving disable, halt and stop reqs
    // Mask set above, nothing to do
    // reqMask := MACM_DISABLE_MASK + MACM_STOP_MASK + MACM_HALT_MASK;
    ;
  ELSE
    // Move allowed, leave the request
    // Modify the mask set above, and clear the other move requests, preserving disable, halt and stop reqs
    reqMask := reqMask + MACM_RELATIVE_MOVE_MASK;
  END_IF
END_IF

// Move Absolute Request
IF ax.Commands.MoveAbsoluteReq THEN
  ActionChkPermissiveAbs;
  IF (ax.Commands.MoveNotAllowed OR NOT ax.Status.IsHomed OR ax.ForceSetRef) THEN
    // Move not allowed in requested direction or axis is not homed, or it needs to be re-referenced
    // Set the mask to clear the request, preserving disable, halt and stop reqs
    // Mask set above, nothing to do
    // reqMask := MACM_DISABLE_MASK + MACM_STOP_MASK + MACM_HALT_MASK;
    ;
  ELSE
    // Move allowed, leave the request
    // Modify the mask set above, and clear the other move requests, preserving disable, halt and stop reqs
    reqMask := reqMask + MACM_ABSOLUTE_MOVE_MASK;
  END_IF
END_IF

// Clear the requests based on the mask set above
fctClearMotionRequests(_I_ReqMask := reqMask, _IO_Commands := ax.Commands);

// Call motion command to get status and enable the axis
ActionCallMotionFunctions;

// Run the mode mismatch timer if the mode is not ok.
// Assume mode is okay - no modes on this system
tmrModeMismatch(IN:= FALSE);
END_STEP
(* @SFCCOMMENT := 'Power On and wait for a command' *)
ENTRY_ACTION
// Set the state
ax.SMState:= GAMOT_ASMS_ENABLED;

// reset the mode mismatch timer
tmrModeMismatch(IN:= FALSE);
END_ACTION
TRANSITION FROM Step_Enabled TO Step_Ignore_Axis:=
ax.Ignore
END_TRANSITION
(* @SFCISJUMP := 'Step_Ignore_Axis' *)
TRANSITION Invalid Status FROM Step_Enabled TO Step_AxisValid_Check:=
ax.statusFpMpAxisBasic.StatusId = mcAXIS_ERR_ACTIVATION OR
ax.statusFpMpAxisBasic.StatusId = mcAXIS_ERR_MPLINK_NULL OR
ax.statusFpMpAxisBasic.StatusId = mcAXIS_ERR_MPLINK_INVALID OR
ax.statusFpMpAxisBasic.StatusId = mcAXIS_ERR_MPLINK_CHANGED OR
ax.statusFpMpAxisBasic.StatusId = mcAXIS_ERR_MPLINK_CORRUPT OR
ax.statusFpMpAxisBasic.StatusId = mcAXIS_ERR_MPLINK_IN_USE OR
ax.statusFpMpAxisBasic.StatusId = mcAXIS_ERR_PAR_NULL

END_TRANSITION
(* @SFCISJUMP := 'Step_AxisValid_Check' *)
TRANSITION global or axis stop req FROM Step_Enabled TO Step_StopReq:=
// Global or axis Stop Request
// Note these may be attempted even if there is an error
// as errors are not checked before this.
ax.Commands.StopReq OR gMotionCommands.StopReq
END_TRANSITION
STEP Step_StopReq:
// From the stop state you can only leave with a stop reset req, or an error of some sort.
// Excert the stop cmd, the enable cmd, and preserve the stop reset req.
// Preserve the disable request -- this allows disableing after stopping.
ax.Commands.EnableCmd := TRUE;
ax.Commands.StopCmd := TRUE;
fctClearMotionCommands(_I_CmdMask := MACM_ENABLE_MASK + MACM_STOP_MASK, _IO_Commands := ax.Commands);
fctClearMotionRequests(_I_ReqMask := MACM_DISABLE_MASK + MACM_STOP_RESET_MASK, _IO_Commands := ax.Commands);

// Set the stop params using the values in the move params.
// Stop and halt are now implemented in a similar way, but Stop uses max decel, and forces a reset after.
// For a stop, until the reset is received, the stop cmd is exerted, and the axis state will stay in the Stopping state.
// Halt uses normal decel, and transitions back to enable after the axis is stopped.
// Halt is meant for a 'normal' process stop. Stop is meant for cases where intervention (a reset) should be forced.
ax.MoveParameters.StopParams.Deceleration := ax.MoveParameters.DecelMax;
ax.MoveParameters.StopParams.Jerk := 0.0;
// Stop at position isn't needed, but expose the params here and guess at logical defaults in case they are needed in the future.
ax.MoveParameters.StopParams.StopAtPosition.Activate := FALSE;
ax.MoveParameters.StopParams.StopAtPosition.Deceleration := ax.MoveParameters.Deceleration;
ax.MoveParameters.StopParams.StopAtPosition.Position := ax.MoveParameters.Position;

// Call motion command to get status, and issue the stop and enable commands.
ActionCallMotionFunctions;
END_STEP
ENTRY_ACTION
// Set the state
ax.SMState:= GAMOT_ASMS_STOP;
END_ACTION
TRANSITION Invalid Status FROM Step_StopReq TO Step_AxisValid_Check:=
ax.statusFpMpAxisBasic.StatusId = mcAXIS_ERR_ACTIVATION OR
ax.statusFpMpAxisBasic.StatusId = mcAXIS_ERR_MPLINK_NULL OR
ax.statusFpMpAxisBasic.StatusId = mcAXIS_ERR_MPLINK_INVALID OR
ax.statusFpMpAxisBasic.StatusId = mcAXIS_ERR_MPLINK_CHANGED OR
ax.statusFpMpAxisBasic.StatusId = mcAXIS_ERR_MPLINK_CORRUPT OR
ax.statusFpMpAxisBasic.StatusId = mcAXIS_ERR_MPLINK_IN_USE OR
ax.statusFpMpAxisBasic.StatusId = mcAXIS_ERR_PAR_NULL
END_TRANSITION
(* @SFCISJUMP := 'Step_AxisValid_Check' *)
TRANSITION error FROM Step_StopReq TO Step_Error_Stop:=
// Valid status, but an error
ax.statusFpMpAxisBasic.StatusId = mcAXIS_ERR_PLC_OPEN OR
ax.statusFpMpAxisBasic.Error OR
ax.Status.PlcOpenState = mcAXIS_ERRORSTOP OR
ax.Status.PlcOpenState = mcAXIS_INVALID_CONFIGURATION

END_TRANSITION
(* @SFCISJUMP := 'Step_Error_Stop' *)
TRANSITION stopped, reset req, no errors FROM Step_StopReq TO Step_Stop_Reset:=
// No errors and drive is stopped, in the standstill state, and a reset req was made
(ax.statusFpMpAxisBasic.StatusId = mcAXIS_NO_ERROR OR
ax.statusFpMpAxisBasic.StatusId = mcAXIS_WRN_PLC_OPEN OR
ax.statusFpMpAxisBasic.StatusId = mcAXIS_WRN_MULTIPLE_COMMAND) AND
NOT ax.statusFpMpAxisBasic.Error AND
ax.Status.PlcOpenState = mcAXIS_STOPPING AND // state will remain in Stopping unitl stop cmd is removed
ax.Status.IsStopped AND
ax.Commands.StopResetReq
END_TRANSITION
STEP Step_Stop_Reset:
// Clear the commands and requests, but preserve the enable cmd to keep from
// turning off the axis.
ax.Commands.EnableCmd := TRUE;
fctClearMotionCommands(_I_CmdMask := MACM_ENABLE_MASK, _IO_Commands := ax.Commands);
fctClearMotionRequests(_I_ReqMask := MACM_NOMASK, _IO_Commands := ax.Commands);

// Call motion command to get status, and issue the enable command.
ActionCallMotionFunctions;
END_STEP
ENTRY_ACTION
// Set the state
ax.SMState:= GAMOT_ASMS_STOP_RESET;
END_ACTION
TRANSITION FROM Step_Stop_Reset TO Step_Enabled:=
TRUE
END_TRANSITION
(* @SFCISJUMP := 'Step_Enabled' *)
TRANSITION global or axis halt req FROM Step_Enabled TO Step_HaltReq:=
// Global or axis Stop Request
// Note these may be attempted even if there is an error
// as errors are not checked before this.
ax.Commands.HaltReq OR gMotionCommands.HaltReq

END_TRANSITION
STEP Step_HaltReq:
// From the halt state you can only leave with an error of some sort, or it leaves once the axis stops and goes to the enabled state.
// Excert the stop cmd, and the the enable cmd.
// Preserve the disable request -- this allows disableing after stopping.
ax.Commands.EnableCmd := TRUE;
ax.Commands.StopCmd := TRUE;
fctClearMotionCommands(_I_CmdMask := MACM_ENABLE_MASK + MACM_STOP_MASK, _IO_Commands := ax.Commands);
fctClearMotionRequests(_I_ReqMask := MACM_DISABLE_MASK, _IO_Commands := ax.Commands);

// Set the stop params using the values in the move params.
// Stop and halt are now implemented in a similar way, but Stop uses max decel, and forces a reset after.
// For a stop, until the reset is received, the stop cmd is exerted, and the axis state will stay in the Stopping state.
// Halt uses normal decel, and transitions back to enable after the axis is stopped.
// Halt is meant for a 'normal' process stop. Stop is meant for cases where intervention (a reset) should be forced.
ax.MoveParameters.StopParams.Deceleration := ax.MoveParameters.Deceleration;
ax.MoveParameters.StopParams.Jerk := 0.0;
// Stop at position isn't needed, but expose the params here and guess at logical defaults in case they are needed in the future.
ax.MoveParameters.StopParams.StopAtPosition.Activate := FALSE;
ax.MoveParameters.StopParams.StopAtPosition.Deceleration := ax.MoveParameters.Deceleration;
ax.MoveParameters.StopParams.StopAtPosition.Position := ax.MoveParameters.Position;

// Call motion command to get status, and issue the stop and enable commands.
ActionCallMotionFunctions;
END_STEP
ENTRY_ACTION
// Set the state
ax.SMState:= GAMOT_ASMS_HALT;
END_ACTION
EXIT_ACTION
// Clear the commands and requests, but preserve the enable cmd to keep from
// turning off the axis.
// Preserve the disable request -- this allows disableing after stopping.
ax.Commands.EnableCmd := TRUE;
fctClearMotionCommands(_I_CmdMask := MACM_ENABLE_MASK, _IO_Commands := ax.Commands);
fctClearMotionRequests(_I_ReqMask := MACM_DISABLE_MASK, _IO_Commands := ax.Commands);
// Call motion command to get status, and issue the enable command.
ActionCallMotionFunctions;
END_ACTION
TRANSITION Invalid Status FROM Step_HaltReq TO Step_AxisValid_Check:=
ax.statusFpMpAxisBasic.StatusId = mcAXIS_ERR_ACTIVATION OR
ax.statusFpMpAxisBasic.StatusId = mcAXIS_ERR_MPLINK_NULL OR
ax.statusFpMpAxisBasic.StatusId = mcAXIS_ERR_MPLINK_INVALID OR
ax.statusFpMpAxisBasic.StatusId = mcAXIS_ERR_MPLINK_CHANGED OR
ax.statusFpMpAxisBasic.StatusId = mcAXIS_ERR_MPLINK_CORRUPT OR
ax.statusFpMpAxisBasic.StatusId = mcAXIS_ERR_MPLINK_IN_USE OR
ax.statusFpMpAxisBasic.StatusId = mcAXIS_ERR_PAR_NULL
END_TRANSITION
(* @SFCISJUMP := 'Step_AxisValid_Check' *)
TRANSITION error FROM Step_HaltReq TO Step_Error_Stop:=
// Valid status, but an error
ax.statusFpMpAxisBasic.StatusId = mcAXIS_ERR_PLC_OPEN OR
ax.statusFpMpAxisBasic.Error OR
ax.Status.PlcOpenState = mcAXIS_ERRORSTOP OR
ax.Status.PlcOpenState = mcAXIS_INVALID_CONFIGURATION
END_TRANSITION
(* @SFCISJUMP := 'Step_Error_Stop' *)
TRANSITION axis stopped, no errors FROM Step_HaltReq TO Step_Enabled:=
// No errors and drive is at a standstill.
(ax.statusFpMpAxisBasic.StatusId = mcAXIS_NO_ERROR OR
ax.statusFpMpAxisBasic.StatusId = mcAXIS_WRN_PLC_OPEN OR
ax.statusFpMpAxisBasic.StatusId = mcAXIS_WRN_MULTIPLE_COMMAND) AND
NOT ax.statusFpMpAxisBasic.Error AND
ax.Status.PlcOpenState = mcAXIS_STOPPING AND // state will remain in Stopping unitl stop cmd is removed
ax.Status.IsStopped  // once stoped, we can leave
END_TRANSITION
(* @SFCISJUMP := 'Step_Enabled' *)
TRANSITION valid and global or axis disable req FROM Step_Enabled TO Step_Disabled:=
// Valid status (allow the couple axis warnings), no errors and global or axis disable req
(ax.statusFpMpAxisBasic.StatusId = mcAXIS_NO_ERROR OR
ax.statusFpMpAxisBasic.StatusId = mcAXIS_WRN_PLC_OPEN OR
ax.statusFpMpAxisBasic.StatusId = mcAXIS_WRN_MULTIPLE_COMMAND) AND
NOT ax.statusFpMpAxisBasic.Error AND
(ax.Commands.DisableReq OR gMotionCommands.DisableReq)
END_TRANSITION
(* @SFCISJUMP := 'Step_Disabled' *)
TRANSITION valid but error FROM Step_Enabled TO Step_Error_Stop:=
// Valid status, but an error
ax.statusFpMpAxisBasic.StatusId = mcAXIS_ERR_PLC_OPEN OR
ax.statusFpMpAxisBasic.Error OR
ax.Status.PlcOpenState = mcAXIS_ERRORSTOP OR
ax.Status.PlcOpenState = mcAXIS_INVALID_CONFIGURATION
END_TRANSITION
STEP Step_Error_Stop:
// Exert a stop command and preserve the enable command.
// The axis may or may not be enabled (powered) depending on the error,
// but if it is enabled, don't presume we want it disabled.
// Clear the requests.
ax.Commands.StopCmd := TRUE;
fctClearMotionCommands(_I_CmdMask := MACM_ENABLE_MASK + MACM_STOP_MASK, _IO_Commands := ax.Commands);
fctClearMotionRequests(_I_ReqMask := MACM_NOMASK, _IO_Commands := ax.Commands);

// Set the stop params using the values in the move params.
// Stop and halt are now implemented in a similar way, but Stop uses max decel, and forces a reset after.
// Halt uses normal decel, and transitions back to enable after the axis is stopped.
// Halt is meant for a 'normal' process stop. Stop is meant for cases where intervention should be forced.
ax.MoveParameters.StopParams.Deceleration := ax.MoveParameters.DecelMax;
ax.MoveParameters.StopParams.Jerk := 0.0;
// Stop at position isn't needed, but expose the params here and guess at logical defaults in case they are needed in the future.
ax.MoveParameters.StopParams.StopAtPosition.Activate := FALSE;
ax.MoveParameters.StopParams.StopAtPosition.Deceleration := ax.MoveParameters.Deceleration;
ax.MoveParameters.StopParams.StopAtPosition.Position := ax.MoveParameters.Position;

// Call motion command to get status, and issue the stop and possibly enable commands.
ActionCallMotionFunctions;
END_STEP
ENTRY_ACTION
// Set the state
ax.SMState:= GAMOT_ASMS_ERROR_STOP;
END_ACTION
EXIT_ACTION
// Shut off the stop command
ax.Commands.StopReq:= FALSE;
END_ACTION
TRANSITION Stop Cmd is done or in error FROM Step_Error_Stop TO Step_Error_DrvRstWait:=
// Stop command done or an error, or axis was disabled due to error
ax.Status.PlcOpenState = mcAXIS_STANDSTILL OR
ax.Status.PlcOpenState = mcAXIS_ERRORSTOP OR
ax.Status.PlcOpenState = mcAXIS_DISABLED

END_TRANSITION
STEP Step_Error_DrvRstWait:
// Drive is stopped and is (was) in error.
// The axis may or may not be enabled (powered) depending on the error,
// but if it is enabled, don't presume we want it disabled.
// We wait here for a drive reset request or a disable request.
// Preserve the drive reset and disable requests, but clear the others
fctClearMotionCommands(_I_CmdMask := MACM_ENABLE_MASK, _IO_Commands := ax.Commands);
fctClearMotionRequests(_I_ReqMask := MACM_DISABLE_MASK + MACM_DRIVE_RESET_MASK, _IO_Commands := ax.Commands);

// Call motion command to get status, and disable the drive.
ActionCallMotionFunctions;

// Run a timer to force the step to be active for a minimum time
tmrDriveReset(IN:= TRUE, PT:= T#500ms);

END_STEP
ENTRY_ACTION
// Set the state
ax.SMState:= GAMOT_ASMS_ERROR_DRVRSTWAIT;

// Reset the wait timer
tmrDriveReset(IN:= FALSE);
END_ACTION
TRANSITION drive reset req FROM Step_Error_DrvRstWait TO Step_Error_DriveReset:=
// Drive reset req received and hold time is satisfied
ax.Commands.DriveResetReq AND
tmrDriveReset.Q
END_TRANSITION
TRANSITION Drive disable req FROM Step_Error_DrvRstWait TO Step_Error_Disable:=
// Drive disable req and hold time is satisfied
ax.Commands.DisableReq AND
tmrDriveReset.Q
END_TRANSITION
STEP Step_Error_Disable:
// Clear the enable command, and the drive will be disabled.

// Clear all the commands, but specifically the Enable Cmd to power off the axis.
// Clear all the requests.
fctClearMotionCommands(_I_CmdMask := MACM_NOMASK, _IO_Commands := ax.Commands);
fctClearMotionRequests(_I_ReqMask := MACM_NOMASK, _IO_Commands := ax.Commands);

// Call motion command to get status, and issue the (false) enable cmd
ActionCallMotionFunctions;

// Run a timer to force the step to be active for a minimum time
tmrDriveReset(IN:= TRUE, PT:= T#500ms);

END_STEP
ENTRY_ACTION
// Set the state
ax.SMState:= GAMOT_ASMS_ERROR_DISABLE;

// Reset the wait timer
tmrDriveReset(IN:= FALSE);
END_ACTION
TRANSITION hold time done FROM Step_Error_Disable TO Step_Error_DrvRstWait:=
// Hold time is satisfied. Ignore states as we don't want to get stuck here.
tmrDriveReset.Q
END_TRANSITION
(* @SFCISJUMP := 'Step_Error_DrvRstWait' *)
STEP Step_Error_DriveReset:
// Exert the drive reset cmd
// The axis may or may not be enabled (powered) depending on the error,
// but if it is enabled, don't presume we want it disabled, so honor the enable cmd if present.
// Clear the requests
ax.Commands.DriveResetCmd := TRUE;
fctClearMotionCommands(_I_CmdMask := MACM_ENABLE_MASK + MACM_DRIVE_RESET_MASK, _IO_Commands := ax.Commands);
fctClearMotionRequests(_I_ReqMask := MACM_NOMASK, _IO_Commands := ax.Commands);

// Call motion command to get status, and issue the drive reset command
ActionCallMotionFunctions;

END_STEP
ENTRY_ACTION
// Set the state
ax.SMState:= GAMOT_ASMS_ERROR_DRVRST;
END_ACTION
EXIT_ACTION
// Clear the command
ax.Commands.DriveResetCmd := FALSE;
END_ACTION
TRANSITION Invalid Status FROM Step_Error_DriveReset TO Step_AxisValid_Check:=
ax.statusFpMpAxisBasic.StatusId = mcAXIS_ERR_ACTIVATION OR
ax.statusFpMpAxisBasic.StatusId = mcAXIS_ERR_MPLINK_NULL OR
ax.statusFpMpAxisBasic.StatusId = mcAXIS_ERR_MPLINK_INVALID OR
ax.statusFpMpAxisBasic.StatusId = mcAXIS_ERR_MPLINK_CHANGED OR
ax.statusFpMpAxisBasic.StatusId = mcAXIS_ERR_MPLINK_CORRUPT OR
ax.statusFpMpAxisBasic.StatusId = mcAXIS_ERR_MPLINK_IN_USE OR
ax.statusFpMpAxisBasic.StatusId = mcAXIS_ERR_PAR_NULL

END_TRANSITION
(* @SFCISJUMP := 'Step_AxisValid_Check' *)
TRANSITION error FROM Step_Error_DriveReset TO Step_Error_DrvRstWait:=
// Valid status, but an error
ax.statusFpMpAxisBasic.StatusId = mcAXIS_ERR_PLC_OPEN OR
ax.statusFpMpAxisBasic.Error OR
ax.Status.PlcOpenState = mcAXIS_ERRORSTOP OR
ax.Status.PlcOpenState = mcAXIS_INVALID_CONFIGURATION

END_TRANSITION
(* @SFCISJUMP := 'Step_Error_DrvRstWait' *)
TRANSITION valid, no errors, drive in error stop FROM Step_Error_DriveReset TO Step_Error_DrvRstWait:=
// Valid status (allow the couple axis warnings), and no errors,
// but drive is in ErrorStop. It shouldn't be, but if it is
// the reset didn't work. Go back to DriveResetWait
(ax.statusFpMpAxisBasic.StatusId = mcAXIS_NO_ERROR OR
ax.statusFpMpAxisBasic.StatusId = mcAXIS_WRN_PLC_OPEN OR
ax.statusFpMpAxisBasic.StatusId = mcAXIS_WRN_MULTIPLE_COMMAND) AND
NOT ax.statusFpMpAxisBasic.Error AND
ax.Status.PlcOpenState = mcAXIS_ERRORSTOP

END_TRANSITION
(* @SFCISJUMP := 'Step_Error_DrvRstWait' *)
TRANSITION valid, no errors, drive (powered) in standstill FROM Step_Error_DriveReset TO Step_Enabled:=
// Valid status (allow the couple axis warnings), and no errors,
// and drive in enabled and in standstill
(ax.statusFpMpAxisBasic.StatusId = mcAXIS_NO_ERROR OR
ax.statusFpMpAxisBasic.StatusId = mcAXIS_WRN_PLC_OPEN OR
ax.statusFpMpAxisBasic.StatusId = mcAXIS_WRN_MULTIPLE_COMMAND) AND
NOT ax.statusFpMpAxisBasic.Error AND
ax.Status.PlcOpenState = mcAXIS_STANDSTILL

END_TRANSITION
(* @SFCISJUMP := 'Step_Enabled' *)
TRANSITION valid, no errors, drive disabled FROM Step_Error_DriveReset TO Step_Disabled:=
// Valid status (allow the couple axis warnings), and no errors,
// and drive in disabled
(ax.statusFpMpAxisBasic.StatusId = mcAXIS_NO_ERROR OR
ax.statusFpMpAxisBasic.StatusId = mcAXIS_WRN_PLC_OPEN OR
ax.statusFpMpAxisBasic.StatusId = mcAXIS_WRN_MULTIPLE_COMMAND) AND
NOT ax.statusFpMpAxisBasic.Error AND
ax.Status.PlcOpenState = mcAXIS_DISABLED

END_TRANSITION
(* @SFCISJUMP := 'Step_Disabled' *)
TRANSITION Mode problem FROM Step_Enabled TO Step_Disabled:=
// mode mismatch timer times out
tmrModeMismatch.Q
END_TRANSITION
(* @SFCISJUMP := 'Step_Disabled' *)
TRANSITION valid axis, engage as a slave FROM Step_Enabled TO Step_EngageReq:=
// Valid status (allow the couple axis warnings), no errors and engaged as a slave
(ax.statusFpMpAxisBasic.StatusId = mcAXIS_NO_ERROR OR
ax.statusFpMpAxisBasic.StatusId = mcAXIS_WRN_PLC_OPEN OR
ax.statusFpMpAxisBasic.StatusId = mcAXIS_WRN_MULTIPLE_COMMAND) AND
NOT ax.statusFpMpAxisBasic.Error AND
ax.Status.PlcOpenState = mcAXIS_SYNCHRONIZED_MOTION
END_TRANSITION
STEP Step_EngageReq:
// An engage request was made. From here you can:
// Engage as a slave or due to move permissives or some other request,
// disengage, react to errors or get to the disengaged state.
// TODO: Figure out if any reaction to MoveNotAllowed or a bad Engage as Slave permissive is needed.
// Other moves (jog, abs, rel) are not allowed.
// Note the halt request is not acted on while synchronized to the master, as this axis will follow the axis, and presumalbly the master will stop if it needs to.
// The halt request, however, is allowed to stand, so if set, the axis will stop after being disengaged.
// Note that the disable, halt, and stop requests are allowed to stand, but it will be handled by transitioning to disengaged and then onto ready, and then stopped.
// NOTE: It is probably the case for coordinated moves that the slave be engaged as a move permissive for the master, so the above requests should probably stop the master.

// Check positive and negative move permissives and allowable position range
ActionChkPermissiveEngagedSlave;

// If a move is allowed, allow the axis to be engaged as a slave, otherwise don't
IF NOT ax.Commands.MoveNotAllowed THEN
  // Move allowed, so engaging is allowed - set the command
  // TODO: Anything to do? Action is on the master side, so slave may not need to do anything
  ;
ELSE
  // Move not allowed.
  // TODO: Anything to do? Action is on the master side, so slave may not need to do anything
  ;
END_IF;

// If the parameter is set, then set the halt request. Halt won't have an effect while
//engaged, but the axis will be halted after disengaging.
ax.Commands.HaltReq:= ax.MoveParameters.HaltOnSlaveDisengage;

ax.Commands.EnableCmd := TRUE; // Keep from turning off the axis.
fctClearMotionCommands(_I_CmdMask := MACM_ENABLE_MASK, _IO_Commands := ax.Commands);
reqMask := MACM_DISABLE_MASK + MACM_HALT_MASK + MACM_STOP_MASK;
fctClearMotionRequests(_I_ReqMask := reqMask, _IO_Commands := ax.Commands);

// Call motion command to get status, and issue the enable, and hopefully the engage slave cmd.
ActionCallMotionFunctions;

END_STEP
ENTRY_ACTION
// Set the state
ax.SMState:= GAMOT_ASMS_ENGAGED_AS_SLAVE;
END_ACTION
TRANSITION FROM Step_EngageReq TO Step_Ignore_Axis:=
ax.Ignore
END_TRANSITION
(* @SFCISJUMP := 'Step_Ignore_Axis' *)
TRANSITION Invalid status FROM Step_EngageReq TO Step_Disengage:=
ax.statusFpMpAxisBasic.StatusId = mcAXIS_ERR_ACTIVATION OR
ax.statusFpMpAxisBasic.StatusId = mcAXIS_ERR_MPLINK_NULL OR
ax.statusFpMpAxisBasic.StatusId = mcAXIS_ERR_MPLINK_INVALID OR
ax.statusFpMpAxisBasic.StatusId = mcAXIS_ERR_MPLINK_CHANGED OR
ax.statusFpMpAxisBasic.StatusId = mcAXIS_ERR_MPLINK_CORRUPT OR
ax.statusFpMpAxisBasic.StatusId = mcAXIS_ERR_MPLINK_IN_USE OR
ax.statusFpMpAxisBasic.StatusId = mcAXIS_ERR_PAR_NULL

END_TRANSITION
TRANSITION global or axis stop req FROM Step_EngageReq TO Step_Disengage:=
// Global or axis Stop Request
// Note these may be attempted even if there is an error
// as errors are not checked before this.
ax.Commands.StopReq OR gMotionCommands.StopReq

END_TRANSITION
TRANSITION valid and global or axis disable req FROM Step_EngageReq TO Step_Disengage:=
// Valid status (allow the couple axis warnings), no errors and global or axis disable req
(ax.statusFpMpAxisBasic.StatusId = mcAXIS_NO_ERROR OR
ax.statusFpMpAxisBasic.StatusId = mcAXIS_WRN_PLC_OPEN OR
ax.statusFpMpAxisBasic.StatusId = mcAXIS_WRN_MULTIPLE_COMMAND) AND
NOT ax.statusFpMpAxisBasic.Error AND
(ax.Commands.DisableReq OR gMotionCommands.DisableReq)
END_TRANSITION
TRANSITION Disengaged as slave FROM Step_EngageReq TO Step_Disengage:=
// Valid status (allow the couple axis warnings), no errors, but not in sync motion any more
(ax.statusFpMpAxisBasic.StatusId = mcAXIS_NO_ERROR OR
ax.statusFpMpAxisBasic.StatusId = mcAXIS_WRN_PLC_OPEN OR
ax.statusFpMpAxisBasic.StatusId = mcAXIS_WRN_MULTIPLE_COMMAND) AND
NOT ax.statusFpMpAxisBasic.Error AND
ax.Status.PlcOpenState <> mcAXIS_SYNCHRONIZED_MOTION
END_TRANSITION
TRANSITION valid but error FROM Step_EngageReq TO Step_Disengage:=
// Axis is valid, but there are errors
ax.statusFpMpAxisBasic.StatusId = mcAXIS_ERR_PLC_OPEN OR
ax.statusFpMpAxisBasic.Error OR
ax.Status.PlcOpenState = mcAXIS_ERRORSTOP OR
ax.Status.PlcOpenState = mcAXIS_INVALID_CONFIGURATION
END_TRANSITION
STEP Step_Disengage:
// The axis was engaged as a slave but is now disengaged,
// either because of a request or error.
// Excert the enable command and the disengage command.
// Allow the disable, halt, and stop requests to stand

// TODO: Deal with MpAxisCoupling
// TODO: Deal with whether or not motion should stop or continue.
// NOTE: It is probably the case for coordinated moves that the slave be engaged as a move permissive for the master, so the above requests should probably stop the master.

ax.Commands.EnableCmd := TRUE;
fctClearMotionCommands(_I_CmdMask := MACM_ENABLE_MASK, _IO_Commands := ax.Commands);
fctClearMotionRequests(_I_ReqMask := MACM_DISABLE_MASK + MACM_HALT_MASK + MACM_STOP_MASK, _IO_Commands := ax.Commands);

// Call motion command to get status, and issue the enable and disengage commands.
// TODO: Implement Axis Coupling
ActionCallMotionFunctions;

END_STEP
ENTRY_ACTION
// Set the state
ax.SMState:= GAMOT_ASMS_DISENGAGE_AS_SLAVE;
END_ACTION
TRANSITION FROM Step_Disengage TO Step_Enabled:=
TRUE
END_TRANSITION
(* @SFCISJUMP := 'Step_Enabled' *)
TRANSITION valid, home req FROM Step_Enabled TO Step_HomeReq:=
// Valid status (allow the couple axis warnings), no errors and home req
(ax.statusFpMpAxisBasic.StatusId = mcAXIS_NO_ERROR OR
ax.statusFpMpAxisBasic.StatusId = mcAXIS_WRN_PLC_OPEN OR
ax.statusFpMpAxisBasic.StatusId = mcAXIS_WRN_MULTIPLE_COMMAND) AND
NOT ax.statusFpMpAxisBasic.Error AND
ax.Commands.HomeReq
END_TRANSITION
STEP Step_HomeReq:
// From here, try to home the axis. It will either have an error or become homed.
// Preserve the enable bit so the axis isn't forced off.
// Turn off the other requests.
ax.Commands.HomeCmd := TRUE;
fctClearMotionCommands(_I_CmdMask := MACM_ENABLE_MASK + MACM_HOME_MASK, _IO_Commands := ax.Commands);
fctClearMotionRequests(_I_ReqMask := MACM_NOMASK, _IO_Commands := ax.Commands);

// Call motion command to get status, and issue the home command, and possibly the enable command.
ActionCallMotionFunctions;

// Run the timer which holds here for a bit
tmrHomeMinimum(IN:= TRUE);
END_STEP
ENTRY_ACTION
// Set the state
ax.SMState:= GAMOT_ASMS_HOME_REQ;
// reset the timer
tmrHomeMinimum(IN:= FALSE, PT:= T#100ms);
END_ACTION
TRANSITION error FROM Step_HomeReq TO Step_Error_Stop:=
// Valid status, but an error
ax.statusFpMpAxisBasic.StatusId = mcAXIS_ERR_PLC_OPEN OR
ax.statusFpMpAxisBasic.Error OR
ax.Status.PlcOpenState = mcAXIS_ERRORSTOP OR
ax.Status.PlcOpenState = mcAXIS_INVALID_CONFIGURATION

END_TRANSITION
(* @SFCISJUMP := 'Step_Error_Stop' *)
TRANSITION homing FROM Step_HomeReq TO StepHoming:=
// Timer check ensures homing command was at least received.
tmrHomeMinimum.Q AND
(ax.Status.AxisDiagnostics.ExecutingCommand = mcAXIS_CMD_HOMING OR
ax.Status.PlcOpenState = mcAXIS_HOMING OR
ax.Status.PlcOpenState = mcAXIS_DISABLED OR
ax.Status.PlcOpenState = mcAXIS_STANDSTILL OR
ax.Status.PlcOpenState = mcAXIS_STOPPING)
END_TRANSITION
STEP StepHoming:
// Continue the home command
// Preserve the enable bit so the axis isn't forced off.
// Turn off the other requests.
ax.Commands.HomeCmd := TRUE;
fctClearMotionCommands(_I_CmdMask := MACM_ENABLE_MASK + MACM_HOME_MASK, _IO_Commands := ax.Commands);
fctClearMotionRequests(_I_ReqMask := MACM_NOMASK, _IO_Commands := ax.Commands);

// Call motion command to get status, and issue the home command, and possibly the enable command.
ActionCallMotionFunctions;
END_STEP
ENTRY_ACTION
// Set the state
ax.SMState:= GAMOT_ASMS_HOMING;
END_ACTION
EXIT_ACTION
// Make sure command is off on exit
ax.Commands.HomeCmd:= FALSE;
END_ACTION
TRANSITION error FROM StepHoming TO Step_Error_Stop:=
// Valid status, but an error
ax.statusFpMpAxisBasic.StatusId = mcAXIS_ERR_PLC_OPEN OR
ax.statusFpMpAxisBasic.Error OR
ax.Status.PlcOpenState = mcAXIS_ERRORSTOP OR
ax.Status.PlcOpenState = mcAXIS_INVALID_CONFIGURATION

END_TRANSITION
(* @SFCISJUMP := 'Step_Error_Stop' *)
TRANSITION Homed FROM StepHoming TO Step_Homed:=
// Valid status (allow the couple axis warnings), homed, and no errors and disabled or standstill
(ax.statusFpMpAxisBasic.StatusId = mcAXIS_NO_ERROR OR
ax.statusFpMpAxisBasic.StatusId = mcAXIS_WRN_PLC_OPEN OR
ax.statusFpMpAxisBasic.StatusId = mcAXIS_WRN_MULTIPLE_COMMAND) AND
NOT ax.statusFpMpAxisBasic.Error AND
ax.Status.IsHomed AND
(ax.Status.PlcOpenState = mcAXIS_DISABLED OR
ax.Status.PlcOpenState = mcAXIS_STANDSTILL)
END_TRANSITION
STEP Step_Homed:
END_STEP
ENTRY_ACTION
// Set the state
ax.SMState:= GAMOT_ASMS_HOMED;
// Clear the force set ref
ax.ForceSetRef := FALSE;

END_ACTION
TRANSITION Drive disabled FROM Step_Homed TO Step_Disabled:=
// Drive is disabled after homing, so go tho that state
ax.Status.PlcOpenState = mcAXIS_DISABLED
END_TRANSITION
(* @SFCISJUMP := 'Step_Disabled' *)
TRANSITION Drive enabled FROM Step_Homed TO Step_Enabled:=
// Drive is enabled after homing, so go to that state
ax.Status.PlcOpenState = mcAXIS_STANDSTILL
END_TRANSITION
(* @SFCISJUMP := 'Step_Enabled' *)
TRANSITION valid, jog req FROM Step_Enabled TO Step_JogReq:=
// Velocity move or jog positive limit or jog negative limit used in place of jog
FALSE
// Valid status (allow the couple axis warnings), no errors and jog req
// (ax.statusFpMpAxisBasic.AxisError = mcAXIS_NO_ERROR OR
// ax.statusFpMpAxisBasic.AxisError = mcAXIS_WRN_PLC_OPEN OR
// ax.statusFpMpAxisBasic.AxisError = mcAXIS_WRN_MULTIPLE_COMMAND) AND
// NOT ax.statusFpMpAxisBasic.Error AND
// ax.Commands.MoveJogReq
END_TRANSITION
STEP Step_JogReq:
// If the move is allowed, execute the jog command, and keep the enable command or the axis will shut off.
// Preserve the other move commands.  Other move requests will cause a state change.
// Preserve the halt, stop, and disable requests.
ax.Commands.EnableCmd := TRUE;

// Use the move parameter position limits, accel, decel and jerk for the jog
// This way, the application can worry about these values in the
// parameter structure, but not have to worry about the jog limits.
ax.MoveParameters.JogParams.Velocity := ax.MoveParameters.Velocity;
ax.MoveParameters.JogParams.LimitPosition.FirstPosition :=  axPositionLimits.PositionLimitNeg;
ax.MoveParameters.JogParams.LimitPosition.LastPosition :=  axPositionLimits.PositionLimitPos;
ax.MoveParameters.JogParams.Acceleration := ax.MoveParameters.Acceleration;
ax.MoveParameters.JogParams.Deceleration := ax.MoveParameters.Deceleration;
ax.MoveParameters.JogParams.Jerk := ax.MoveParameters.MaxJerk;

// Set the request mask for those requests we know we want to honor.
// This move may or may not be allowed, but since it is a jog, it the request should be maintained,
// and a stop/halt/move/ or other reqeest will clear it.
reqMask := MACM_DISABLE_MASK + MACM_JOG_POSITIVE_MASK + MACM_JOG_NEGATIVE_MASK +
MACM_VELOCITY_MOVE_MASK + MACM_RELATIVE_MOVE_MASK + MACM_ABSOLUTE_MOVE_MASK + MACM_STOP_MASK + MACM_HALT_MASK;

// Check move permissives -- move of undefined length
ActionChkPermissiveContinuous;

// If the move is allowed, set the command, otherwise clear it
IF NOT ax.Commands.MoveNotAllowed THEN
  // Move is allowed.
  // Set the command but don't clear the request -- the jog should continue
  // as long as the request is held
  ax.Commands.MoveJogCmd:= TRUE;
  reqMask := reqMask + MACM_JOG_MASK;
ELSE
  // Move not allowed. Clear the cmd, req, and issue a halt
  ax.Commands.MoveJogReq:= FALSE;
  ax.Commands.MoveJogCmd:= FALSE;
  ax.Commands.HaltReq:= TRUE;
END_IF;

fctClearMotionCommands(_I_CmdMask := MACM_ENABLE_MASK + MACM_JOG_MASK, _IO_Commands := ax.Commands);
fctClearMotionRequests(_I_ReqMask := reqMask, _IO_Commands := ax.Commands);

// Call the motion commands
ActionCallMotionFunctions;

// Run the mode mismatch timer if the mode is not ok.
// Assume mode is okay - no modes on this system
tmrModeMismatch(IN:= FALSE);
END_STEP
ENTRY_ACTION
// Set the state
ax.SMState:= GAMOT_ASMS_JOG;

// Reset the mode check timer
tmrModeMismatch(IN:= FALSE);

END_ACTION
EXIT_ACTION
// Shut off the command and request.
// Unlike other commands, the request for a jog stays on as long as the move is desired.
ax.Commands.MoveJogReq:= FALSE;
ax.Commands.MoveJogCmd:= FALSE;

// Call the motion commands
// Do this here, so the motion function blocks are guaranteed to see a
// falling edge of the command. Unexpected, but not necessarily incorrect
// behavior may result when one command is not ended before another starts.
ActionCallMotionFunctions;

END_ACTION
TRANSITION error FROM Step_JogReq TO Step_Error_Stop:=
// Valid status, but an error
ax.statusFpMpAxisBasic.StatusId = mcAXIS_ERR_PLC_OPEN OR
ax.statusFpMpAxisBasic.Error OR
ax.Status.PlcOpenState = mcAXIS_ERRORSTOP OR
ax.Status.PlcOpenState = mcAXIS_INVALID_CONFIGURATION

END_TRANSITION
(* @SFCISJUMP := 'Step_Error_Stop' *)
TRANSITION stop req FROM Step_JogReq TO Step_StopReq:=
// A global or local stop is requested
ax.Commands.StopReq OR gMotionCommands.StopReq
END_TRANSITION
(* @SFCISJUMP := 'Step_StopReq' *)
TRANSITION mode problem or halt req FROM Step_JogReq TO Step_HaltReq:=
// Mode problem or axis or global halt request
tmrModeMismatch.Q OR
ax.Commands.HaltReq OR gMotionCommands.HaltReq
END_TRANSITION
(* @SFCISJUMP := 'Step_HaltReq' *)
TRANSITION no jog req or other move req FROM Step_JogReq TO Step_Enabled:=
// Valid status (allow the couple axis warnings), no errors and jog req goes away
// or another move request comes in. Note stop and halt are handled separately.
(ax.statusFpMpAxisBasic.StatusId = mcAXIS_NO_ERROR OR
ax.statusFpMpAxisBasic.StatusId = mcAXIS_WRN_PLC_OPEN OR
ax.statusFpMpAxisBasic.StatusId = mcAXIS_WRN_MULTIPLE_COMMAND) AND
(NOT ax.Commands.MoveJogReq OR
ax.Commands.DisableReq OR
ax.Commands.MoveJogPositiveReq OR
ax.Commands.MoveJogNegativeReq OR
ax.Commands.MoveVelocityReq OR
ax.Commands.MoveRelativeReq OR
ax.Commands.MoveAbsoluteReq)
END_TRANSITION
(* @SFCISJUMP := 'Step_Enabled' *)
TRANSITION valid, jog pos limit req FROM Step_Enabled TO Step_JogPosLimitReq:=
// Valid status (allow the couple axis warnings), no errors and jog positive req
(ax.statusFpMpAxisBasic.StatusId = mcAXIS_NO_ERROR OR
ax.statusFpMpAxisBasic.StatusId = mcAXIS_WRN_PLC_OPEN OR
ax.statusFpMpAxisBasic.StatusId = mcAXIS_WRN_MULTIPLE_COMMAND) AND
NOT ax.statusFpMpAxisBasic.Error AND
ax.Commands.MoveJogPositiveReq
END_TRANSITION
STEP Step_JogPosLimitReq:
// If the move is allowed, execute the jog positive limit command, and keep the enable command or the axis will shut off.
// Preserve the other move commands.  Other move requests will cause a state change.
// Preserve the halt, stop, and disable requests.
ax.Commands.EnableCmd := TRUE;

// Use the move parameter position limits, accel, decel and jerk for the jog
// This way, the application can worry about these values in the
// parameter structure, but not have to worry about the jog limits.
ax.MoveParameters.JogParams.Velocity := ax.MoveParameters.Velocity;
ax.MoveParameters.JogParams.LimitPosition.FirstPosition :=  axPositionLimits.PositionLimitNeg;
ax.MoveParameters.JogParams.LimitPosition.LastPosition :=  axPositionLimits.PositionLimitPos;
ax.MoveParameters.JogParams.Acceleration := ax.MoveParameters.Acceleration;
ax.MoveParameters.JogParams.Deceleration := ax.MoveParameters.Deceleration;
ax.MoveParameters.JogParams.Jerk := ax.MoveParameters.MaxJerk;

// Set the request mask for those requests we know we want to honor.
// This move may or may not be allowed, but since it is a jog, it the request should be maintained,
// and a stop/halt/move/ or other reqeest will clear it.
reqMask := MACM_DISABLE_MASK + MACM_JOG_MASK + MACM_JOG_NEGATIVE_MASK +
MACM_VELOCITY_MOVE_MASK + MACM_RELATIVE_MOVE_MASK + MACM_ABSOLUTE_MOVE_MASK + MACM_STOP_MASK + MACM_HALT_MASK;

// Check move permissives -- move of undefined length
ActionChkPermissiveContinuous;

// If the move is allowed, set the command, otherwise clear it
IF NOT ax.Commands.MoveNotAllowed THEN
  // Move is allowed.
  // Set the command but don't clear the request -- the jog should continue
  // as long as the request is held
  ax.Commands.MoveJogPositiveCmd:= TRUE;
  reqMask := reqMask + MACM_JOG_POSITIVE_MASK;
ELSE
  // Move not allowed. Clear the cmd, req, and issue a halt
  ax.Commands.MoveJogPositiveReq:= FALSE;
  ax.Commands.MoveJogPositiveCmd:= FALSE;
  ax.Commands.HaltReq:= TRUE;
END_IF;

fctClearMotionCommands(_I_CmdMask := MACM_ENABLE_MASK + MACM_JOG_POSITIVE_MASK, _IO_Commands := ax.Commands);
fctClearMotionRequests(_I_ReqMask := reqMask, _IO_Commands := ax.Commands);

// Call the motion commands
ActionCallMotionFunctions;

// Run the mode mismatch timer if the mode is not ok.
// Assume mode is okay - no modes on this system
tmrModeMismatch(IN:= FALSE);
END_STEP
ENTRY_ACTION
// Set the state
ax.SMState:= GAMOT_ASMS_JOGPOSLIMIT;

// Reset the mode check timer
tmrModeMismatch(IN:= FALSE);

END_ACTION
EXIT_ACTION
// Shut off the command and request.
// Unlike other commands, the request for a jog stays on as long as the move is desired.
ax.Commands.MoveJogPositiveCmd:= FALSE;
ax.Commands.MoveJogPositiveReq:= FALSE;

// Call the motion commands
// Do this here, so the motion function blocks are guaranteed to see a
// falling edge of the command. Unexpected, but not necessarily incorrect
// behavior may result when one command is not ended before another starts.
ActionCallMotionFunctions;

END_ACTION
TRANSITION error FROM Step_JogPosLimitReq TO Step_Error_Stop:=
// Valid status, but an error
ax.statusFpMpAxisBasic.StatusId = mcAXIS_ERR_PLC_OPEN OR
ax.statusFpMpAxisBasic.Error OR
ax.Status.PlcOpenState = mcAXIS_ERRORSTOP OR
ax.Status.PlcOpenState = mcAXIS_INVALID_CONFIGURATION

END_TRANSITION
(* @SFCISJUMP := 'Step_Error_Stop' *)
TRANSITION stop req FROM Step_JogPosLimitReq TO Step_StopReq:=
// A global or local stop is requested
ax.Commands.StopReq OR gMotionCommands.StopReq
END_TRANSITION
(* @SFCISJUMP := 'Step_StopReq' *)
TRANSITION mode problem or halt req FROM Step_JogPosLimitReq TO Step_HaltReq:=
// Mode problem or axis or global halt request
tmrModeMismatch.Q OR
ax.Commands.HaltReq OR gMotionCommands.HaltReq
END_TRANSITION
(* @SFCISJUMP := 'Step_HaltReq' *)
TRANSITION No jog pos limit req or othe rmove req FROM Step_JogPosLimitReq TO Step_Enabled:=
// Valid status (allow the couple axis warnings), no errors and jog req goes away
// or another move request comes in. Note stop and halt are handled separately.
(ax.statusFpMpAxisBasic.StatusId = mcAXIS_NO_ERROR OR
ax.statusFpMpAxisBasic.StatusId = mcAXIS_WRN_PLC_OPEN OR
ax.statusFpMpAxisBasic.StatusId = mcAXIS_WRN_MULTIPLE_COMMAND) AND
(NOT ax.Commands.MoveJogPositiveReq OR
ax.Commands.DisableReq OR
ax.Commands.MoveJogReq OR
ax.Commands.MoveJogNegativeReq OR
ax.Commands.MoveVelocityReq OR
ax.Commands.MoveRelativeReq OR
ax.Commands.MoveAbsoluteReq)
END_TRANSITION
(* @SFCISJUMP := 'Step_Enabled' *)
TRANSITION valid, jog neg limit req FROM Step_Enabled TO Step_JogNegLimitReq:=
// Valid status (allow the couple axis warnings), no errors and jog negative req
(ax.statusFpMpAxisBasic.StatusId = mcAXIS_NO_ERROR OR
ax.statusFpMpAxisBasic.StatusId = mcAXIS_WRN_PLC_OPEN OR
ax.statusFpMpAxisBasic.StatusId = mcAXIS_WRN_MULTIPLE_COMMAND) AND
NOT ax.statusFpMpAxisBasic.Error AND
ax.Commands.MoveJogNegativeReq
END_TRANSITION
STEP Step_JogNegLimitReq:
// If the move is allowed, execute the jog negative limit command, and keep the enable command or the axis will shut off.
// Preserve the other move commands.  Other move requests will cause a state change.
// Preserve the halt, stop, and disable requests.
ax.Commands.EnableCmd := TRUE;

// Use the move parameter position limits, accel, decel and jerk for the jog
// This way, the application can worry about these values in the
// parameter structure, but not have to worry about the jog limits.
ax.MoveParameters.JogParams.Velocity := ax.MoveParameters.Velocity;
ax.MoveParameters.JogParams.LimitPosition.FirstPosition :=  axPositionLimits.PositionLimitNeg;
ax.MoveParameters.JogParams.LimitPosition.LastPosition :=  axPositionLimits.PositionLimitPos;
ax.MoveParameters.JogParams.Acceleration := ax.MoveParameters.Acceleration;
ax.MoveParameters.JogParams.Deceleration := ax.MoveParameters.Deceleration;
ax.MoveParameters.JogParams.Jerk := ax.MoveParameters.MaxJerk;

// Set the request mask for those requests we know we want to honor.
// This move may or may not be allowed, but since it is a jog, it the request should be maintained,
// and a stop/halt/move/ or other reqeest will clear it.
reqMask := MACM_DISABLE_MASK + MACM_JOG_MASK + MACM_JOG_POSITIVE_MASK +
MACM_VELOCITY_MOVE_MASK + MACM_RELATIVE_MOVE_MASK + MACM_ABSOLUTE_MOVE_MASK + MACM_STOP_MASK + MACM_HALT_MASK;

// Check move permissives -- move of undefined length
ActionChkPermissiveContinuous;

// If the move is allowed, set the command, otherwise clear it
IF NOT ax.Commands.MoveNotAllowed THEN
  // Move is allowed.
  // Set the command but don't clear the request -- the jog should continue
  // as long as the request is held
  ax.Commands.MoveJogNegativeCmd:= TRUE;
  reqMask := reqMask + MACM_JOG_NEGATIVE_MASK;
ELSE
  // Move not allowed. Clear the cmd, req, and issue a halt
  ax.Commands.MoveJogNegativeReq:= FALSE;
  ax.Commands.MoveJogNegativeCmd:= FALSE;
  ax.Commands.HaltReq:= TRUE;
END_IF;

fctClearMotionCommands(_I_CmdMask := MACM_ENABLE_MASK + MACM_JOG_NEGATIVE_MASK, _IO_Commands := ax.Commands);
fctClearMotionRequests(_I_ReqMask := reqMask, _IO_Commands := ax.Commands);

// Call the motion commands
ActionCallMotionFunctions;

// Run the mode mismatch timer if the mode is not ok.
// Assume mode is okay - no modes on this system
tmrModeMismatch(IN:= FALSE);
END_STEP
ENTRY_ACTION
// Set the state
ax.SMState:= GAMOT_ASMS_JOGNEGLIMIT;

// Reset the mode check timer
tmrModeMismatch(IN:= FALSE);

END_ACTION
EXIT_ACTION
// Shut off the command and request.
// Unlike other commands, the request for a jog stays on as long as the move is desired.
ax.Commands.MoveJogNegativeCmd:= FALSE;
ax.Commands.MoveJogNegativeReq:= FALSE;

// Call the motion commands
// Do this here, so the motion function blocks are guaranteed to see a
// falling edge of the command. Unexpected, but not necessarily incorrect
// behavior may result when one command is not ended before another starts.
ActionCallMotionFunctions;

END_ACTION
TRANSITION error FROM Step_JogNegLimitReq TO Step_Error_Stop:=
// Valid status, but an error
ax.statusFpMpAxisBasic.StatusId = mcAXIS_ERR_PLC_OPEN OR
ax.statusFpMpAxisBasic.Error OR
ax.Status.PlcOpenState = mcAXIS_ERRORSTOP OR
ax.Status.PlcOpenState = mcAXIS_INVALID_CONFIGURATION

END_TRANSITION
(* @SFCISJUMP := 'Step_Error_Stop' *)
TRANSITION stop req FROM Step_JogNegLimitReq TO Step_StopReq:=
// A global or local stop is requested
ax.Commands.StopReq OR gMotionCommands.StopReq
END_TRANSITION
(* @SFCISJUMP := 'Step_StopReq' *)
TRANSITION mode problem or halt req FROM Step_JogNegLimitReq TO Step_HaltReq:=
// Mode problem or axis or global halt request
tmrModeMismatch.Q OR
ax.Commands.HaltReq OR gMotionCommands.HaltReq
END_TRANSITION
(* @SFCISJUMP := 'Step_HaltReq' *)
TRANSITION No jog neg limit req or othe rmove req FROM Step_JogNegLimitReq TO Step_Enabled:=
// Valid status (allow the couple axis warnings), no errors and jog req goes away
// or another move request comes in. Note stop and halt are handled separately.
(ax.statusFpMpAxisBasic.StatusId = mcAXIS_NO_ERROR OR
ax.statusFpMpAxisBasic.StatusId = mcAXIS_WRN_PLC_OPEN OR
ax.statusFpMpAxisBasic.StatusId = mcAXIS_WRN_MULTIPLE_COMMAND) AND
(NOT ax.Commands.MoveJogNegativeReq OR
ax.Commands.DisableReq OR
ax.Commands.MoveJogReq OR
ax.Commands.MoveJogPositiveReq OR
ax.Commands.MoveVelocityReq OR
ax.Commands.MoveRelativeReq OR
ax.Commands.MoveAbsoluteReq)
END_TRANSITION
(* @SFCISJUMP := 'Step_Enabled' *)
TRANSITION valid, move velocity FROM Step_Enabled TO Step_MoveVelocityReq:=
// Valid status (allow the couple axis warnings), no errors and jog negative req
(ax.statusFpMpAxisBasic.StatusId = mcAXIS_NO_ERROR OR
ax.statusFpMpAxisBasic.StatusId = mcAXIS_WRN_PLC_OPEN OR
ax.statusFpMpAxisBasic.StatusId = mcAXIS_WRN_MULTIPLE_COMMAND) AND
NOT ax.statusFpMpAxisBasic.Error AND
ax.Commands.MoveVelocityReq
END_TRANSITION
STEP Step_MoveVelocityReq:
// If the move is allowed, execute the move velocity command, and keep the enable command or the axis will shut off.
// Preserve the other move commands.  Other move requests will cause a state change.
// Preserve the halt, stop, and disable requests.
ax.Commands.EnableCmd := TRUE;

// Set the request mask for those requests we know we want to honor.
// This move may or may not be allowed, but since it is a jog, it the request should be maintained,
// and a stop/halt/move/ or other reqeest will clear it.
reqMask := MACM_DISABLE_MASK + MACM_JOG_MASK + MACM_JOG_POSITIVE_MASK + MACM_JOG_NEGATIVE_MASK +
 MACM_RELATIVE_MOVE_MASK + MACM_ABSOLUTE_MOVE_MASK + MACM_STOP_MASK + MACM_HALT_MASK;

// Check move permissives -- move of undefined length
ActionChkPermissiveContinuous;

// If the move is allowed, set the command, otherwise clear it
IF NOT ax.Commands.MoveNotAllowed THEN
  // Move is allowed.
  // Set the command but don't clear the request -- the jog should continue
  // as long as the request is held
  ax.Commands.MoveVelocityCmd:= TRUE;
  reqMask := reqMask + MACM_VELOCITY_MOVE_MASK;
ELSE
  // Move not allowed. Clear the cmd issue a halt
  ax.Commands.MoveVelocityReq:= FALSE;
  ax.Commands.MoveVelocityCmd:= FALSE;
  ax.Commands.HaltReq:= TRUE;
END_IF;

fctClearMotionCommands(_I_CmdMask := MACM_ENABLE_MASK + MACM_VELOCITY_MOVE_MASK, _IO_Commands := ax.Commands);
fctClearMotionRequests(_I_ReqMask := reqMask, _IO_Commands := ax.Commands);

// Call the motion commands
ActionCallMotionFunctions;

// Run the mode mismatch timer if the mode is not ok.
// Assume mode is okay - no modes on this system
tmrModeMismatch(IN:= FALSE);
END_STEP
ENTRY_ACTION
// Set the state
ax.SMState:= GAMOT_ASMS_MOVE_VELOCITY;

// Reset the mode check timer
tmrModeMismatch(IN:= FALSE);

END_ACTION
EXIT_ACTION
// Shut off the command and request.
// Unlike other commands, the request for a velocity move stays on as long as the move is desired.
ax.Commands.MoveVelocityCmd:= FALSE;
ax.Commands.MoveVelocityReq:= FALSE;

// Call the motion commands
// Do this here, so the motion function blocks are guaranteed to see a
// falling edge of the command. Unexpected, but not necessarily incorrect
// behavior may result when one command is not ended before another starts.
ActionCallMotionFunctions;

END_ACTION
TRANSITION error FROM Step_MoveVelocityReq TO Step_Error_Stop:=
// Valid status, but an error
ax.statusFpMpAxisBasic.StatusId = mcAXIS_ERR_PLC_OPEN OR
ax.statusFpMpAxisBasic.Error OR
ax.Status.PlcOpenState = mcAXIS_ERRORSTOP OR
ax.Status.PlcOpenState = mcAXIS_INVALID_CONFIGURATION

END_TRANSITION
(* @SFCISJUMP := 'Step_Error_Stop' *)
TRANSITION stop req FROM Step_MoveVelocityReq TO Step_StopReq:=
// A global or local stop is requested
ax.Commands.StopReq OR gMotionCommands.StopReq
END_TRANSITION
(* @SFCISJUMP := 'Step_StopReq' *)
TRANSITION mode problem or halt req FROM Step_MoveVelocityReq TO Step_HaltReq:=
// Mode problem or axis or global halt request
tmrModeMismatch.Q OR
ax.Commands.HaltReq OR gMotionCommands.HaltReq
END_TRANSITION
(* @SFCISJUMP := 'Step_HaltReq' *)
TRANSITION no vel req or other move req FROM Step_MoveVelocityReq TO Step_Enabled:=
// Valid status (allow the couple axis warnings), no errors and vel req goes away
// or another move request comes in. Note stop and halt are handled separately.
(ax.statusFpMpAxisBasic.StatusId = mcAXIS_NO_ERROR OR
ax.statusFpMpAxisBasic.StatusId = mcAXIS_WRN_PLC_OPEN OR
ax.statusFpMpAxisBasic.StatusId = mcAXIS_WRN_MULTIPLE_COMMAND) AND
(NOT ax.Commands.MoveVelocityReq OR
ax.Commands.DisableReq OR
ax.Commands.MoveJogReq OR
ax.Commands.MoveJogPositiveReq OR
ax.Commands.MoveJogNegativeReq OR
ax.Commands.MoveRelativeReq OR
ax.Commands.MoveAbsoluteReq)
END_TRANSITION
(* @SFCISJUMP := 'Step_Enabled' *)
TRANSITION valid, move rel req FROM Step_Enabled TO Step_MoveRelativeReq:=
// Valid status (allow the couple axis warnings), no errors and jog negative req
(ax.statusFpMpAxisBasic.StatusId = mcAXIS_NO_ERROR OR
ax.statusFpMpAxisBasic.StatusId = mcAXIS_WRN_PLC_OPEN OR
ax.statusFpMpAxisBasic.StatusId = mcAXIS_WRN_MULTIPLE_COMMAND) AND
NOT ax.statusFpMpAxisBasic.Error AND
ax.Commands.MoveRelativeReq
END_TRANSITION
STEP Step_MoveRelativeReq:
// If the move is allowed, execute the move relative command, and keep the enable command or the axis will shut off.
// Preserve the other move commands.  Other move requests will cause a state change.
// Preserve the halt, stop, and disable requests.
ax.Commands.EnableCmd := TRUE;

// Set the request mask for those requests we know we want to honor.
// This move may or may not be allowed, but the request has already been honored, so it can be cleared.
reqMask := MACM_DISABLE_MASK + MACM_JOG_MASK + MACM_JOG_POSITIVE_MASK + MACM_JOG_NEGATIVE_MASK +
MACM_VELOCITY_MOVE_MASK + MACM_ABSOLUTE_MOVE_MASK + MACM_STOP_MASK + MACM_HALT_MASK;

// Check move permissives
ActionChkPermissiveRel;

// If the move is allowed, set the command, otherwise clear it
IF NOT ax.Commands.MoveNotAllowed THEN
  // Move is allowed.
  // Set the command but don't clear the request -- the jog should continue
  // as long as the request is held
  ax.Commands.MoveRelativeCmd:= TRUE;
ELSE
  // Move not allowed. Clear the cmd issue a halt
  ax.Commands.MoveRelativeCmd:= FALSE;
  ax.Commands.HaltReq:= TRUE;
END_IF;

fctClearMotionCommands(_I_CmdMask := MACM_ENABLE_MASK + MACM_RELATIVE_MOVE_MASK, _IO_Commands := ax.Commands);
fctClearMotionRequests(_I_ReqMask := reqMask, _IO_Commands := ax.Commands);

// Call the motion commands
ActionCallMotionFunctions;

// Run the mode mismatch timer if the mode is not ok.
// Assume mode is okay - no modes on this system
tmrModeMismatch(IN:= FALSE);
END_STEP
ENTRY_ACTION
// Set the state
ax.SMState:= GAMOT_ASMS_MOVE_RELATIVE;

// Reset the mode check timer
tmrModeMismatch(IN:= FALSE);

// Take a snapshot of the current position.
// This is to allow permissive checking while on the move
// while supporting a changealbe move window
ax.MoveParameters.PermissiveCheck.StartPosition := ax.Status.Position;
END_ACTION
EXIT_ACTION
// Shut off the command and request.
ax.Commands.MoveRelativeCmd:= FALSE;
ax.Commands.MoveRelativeReq:= FALSE;

// Call the motion commands
// Do this here, so the motion function blocks are guaranteed to see a
// falling edge of the command. Unexpected, but not necessarily incorrect
// behavior may result when one command is not ended before another starts.
ActionCallMotionFunctions;

END_ACTION
TRANSITION error FROM Step_MoveRelativeReq TO Step_Error_Stop:=
// Valid status, but an error
ax.statusFpMpAxisBasic.StatusId = mcAXIS_ERR_PLC_OPEN OR
ax.statusFpMpAxisBasic.Error OR
ax.Status.PlcOpenState = mcAXIS_ERRORSTOP OR
ax.Status.PlcOpenState = mcAXIS_INVALID_CONFIGURATION

END_TRANSITION
(* @SFCISJUMP := 'Step_Error_Stop' *)
TRANSITION stop req FROM Step_MoveRelativeReq TO Step_StopReq:=
// A global or local stop is requested
ax.Commands.StopReq OR gMotionCommands.StopReq
END_TRANSITION
(* @SFCISJUMP := 'Step_StopReq' *)
TRANSITION mode problem or halt req FROM Step_MoveRelativeReq TO Step_HaltReq:=
// Mode problem or axis or global halt request
tmrModeMismatch.Q OR
ax.Commands.HaltReq OR gMotionCommands.HaltReq
END_TRANSITION
(* @SFCISJUMP := 'Step_HaltReq' *)
TRANSITION move done or other move req FROM Step_MoveRelativeReq TO Step_Enabled:=
// Valid status (allow the couple axis warnings), no errors and move is done
// or another move request comes in. Note stop and halt are handled separately.
(ax.statusFpMpAxisBasic.StatusId = mcAXIS_NO_ERROR OR
ax.statusFpMpAxisBasic.StatusId = mcAXIS_WRN_PLC_OPEN OR
ax.statusFpMpAxisBasic.StatusId = mcAXIS_WRN_MULTIPLE_COMMAND) AND
(ax.Status.IsMoveDone AND ax.Status.PlcOpenState = mcAXIS_STANDSTILL) OR
(ax.Commands.DisableReq OR
ax.Commands.MoveJogReq OR
ax.Commands.MoveJogPositiveReq OR
ax.Commands.MoveJogNegativeReq OR
ax.Commands.MoveVelocityReq OR
ax.Commands.MoveAbsoluteReq)
END_TRANSITION
(* @SFCISJUMP := 'Step_Enabled' *)
TRANSITION valid, abs move req FROM Step_Enabled TO Step_MoveAbsoluteReq:=
// Valid status (allow the couple axis warnings), no errors and jog negative req
(ax.statusFpMpAxisBasic.StatusId = mcAXIS_NO_ERROR OR
ax.statusFpMpAxisBasic.StatusId = mcAXIS_WRN_PLC_OPEN OR
ax.statusFpMpAxisBasic.StatusId = mcAXIS_WRN_MULTIPLE_COMMAND) AND
NOT ax.statusFpMpAxisBasic.Error AND
ax.Commands.MoveAbsoluteReq
END_TRANSITION
STEP Step_MoveAbsoluteReq:
// If the move is allowed, execute the move absolute command, and keep the enable command or the axis will shut off.
// Preserve the other move commands.  Other move requests will cause a state change.
// Preserve the halt, stop, and disable requests.
ax.Commands.EnableCmd := TRUE;

// Set the request mask for those requests we know we want to honor.
// This move may or may not be allowed, but the request has already been honored, so it can be cleared.
reqMask := MACM_DISABLE_MASK + MACM_JOG_MASK + MACM_JOG_POSITIVE_MASK + MACM_JOG_NEGATIVE_MASK +
MACM_VELOCITY_MOVE_MASK + MACM_RELATIVE_MOVE_MASK + MACM_STOP_MASK + MACM_HALT_MASK;

// Check move permissives
ActionChkPermissiveAbs;

// If the move is allowed, set the command, otherwise clear it
IF NOT ax.Commands.MoveNotAllowed THEN
  // Move is allowed.
  // Set the command but don't clear the request -- the jog should continue
  // as long as the request is held
  ax.Commands.MoveAbsoluteCmd:= TRUE;
ELSE
  // Move not allowed. Clear the cmd issue a halt
  ax.Commands.MoveAbsoluteCmd:= FALSE;
  ax.Commands.HaltReq:= TRUE;
END_IF;

fctClearMotionCommands(_I_CmdMask := MACM_ENABLE_MASK + MACM_ABSOLUTE_MOVE_MASK, _IO_Commands := ax.Commands);
fctClearMotionRequests(_I_ReqMask := reqMask, _IO_Commands := ax.Commands);

// Call the motion commands
ActionCallMotionFunctions;

// Run the mode mismatch timer if the mode is not ok.
// Assume mode is okay - no modes on this system
tmrModeMismatch(IN:= FALSE);
END_STEP
ENTRY_ACTION
// Set the state
ax.SMState:= GAMOT_ASMS_MOVE_ABSOLUTE;

// Reset the mode check timer
tmrModeMismatch(IN:= FALSE);
END_ACTION
EXIT_ACTION
// Shut off the command and request.
ax.Commands.MoveAbsoluteCmd:= FALSE;
ax.Commands.MoveAbsoluteReq:= FALSE;

// Call the motion commands
// Do this here, so the motion function blocks are guaranteed to see a
// falling edge of the command. Unexpected, but not necessarily incorrect
// behavior may result when one command is not ended before another starts.
ActionCallMotionFunctions;

END_ACTION
TRANSITION error FROM Step_MoveAbsoluteReq TO Step_Error_Stop:=
// Valid status, but an error
ax.statusFpMpAxisBasic.StatusId = mcAXIS_ERR_PLC_OPEN OR
ax.statusFpMpAxisBasic.Error OR
ax.Status.PlcOpenState = mcAXIS_ERRORSTOP OR
ax.Status.PlcOpenState = mcAXIS_INVALID_CONFIGURATION

END_TRANSITION
(* @SFCISJUMP := 'Step_Error_Stop' *)
TRANSITION stop req FROM Step_MoveAbsoluteReq TO Step_StopReq:=
// A global or local stop is requested
ax.Commands.StopReq OR gMotionCommands.StopReq
END_TRANSITION
(* @SFCISJUMP := 'Step_StopReq' *)
TRANSITION mode problem or halt req FROM Step_MoveAbsoluteReq TO Step_HaltReq:=
// Mode problem or axis or global halt request
tmrModeMismatch.Q OR
ax.Commands.HaltReq OR gMotionCommands.HaltReq
END_TRANSITION
(* @SFCISJUMP := 'Step_HaltReq' *)
TRANSITION move done or other move req FROM Step_MoveAbsoluteReq TO Step_Enabled:=
// Valid status (allow the couple axis warnings), no errors and move is done
// or another move request comes in. Note stop and halt are handled separately.
(ax.statusFpMpAxisBasic.StatusId = mcAXIS_NO_ERROR OR
ax.statusFpMpAxisBasic.StatusId = mcAXIS_WRN_PLC_OPEN OR
ax.statusFpMpAxisBasic.StatusId = mcAXIS_WRN_MULTIPLE_COMMAND) AND
(ax.Status.IsMoveDone AND ax.Status.PlcOpenState = mcAXIS_STANDSTILL) OR
(ax.Commands.DisableReq OR
ax.Commands.MoveJogReq OR
ax.Commands.MoveJogPositiveReq OR
ax.Commands.MoveJogNegativeReq OR
ax.Commands.MoveVelocityReq OR
ax.Commands.MoveRelativeReq)
END_TRANSITION
(* @SFCISJUMP := 'Step_Enabled' *)
TRANSITION valid but error FROM Step_AxisValid_Check TO Step_Error_DrvRstWait:=
// Axis is valid, but there are errors
ax.statusFpMpAxisBasic.StatusId = mcAXIS_ERR_PLC_OPEN OR
ax.statusFpMpAxisBasic.Error OR
ax.Status.PlcOpenState = mcAXIS_ERRORSTOP OR
ax.Status.PlcOpenState = mcAXIS_INVALID_CONFIGURATION

END_TRANSITION
(* @SFCISJUMP := 'Step_Error_DrvRstWait' *)
END_PROGRAM
```
